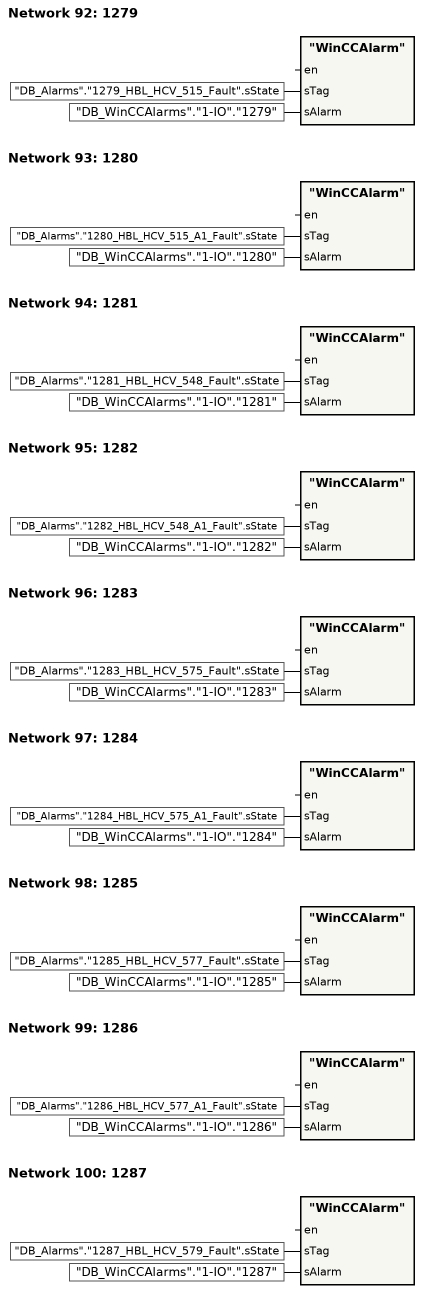
   "WinCCAlarm"(sTag := "DB_Alarms"."1279_HBL_HCV_515_Fault".sState, sAlarm := "DB_WinCCAlarms"."1-IO"."1279");
END_REGION

REGION Network 93: 1280
   "WinCCAlarm"(sTag := "DB_Alarms"."1280_HBL_HCV_515_A1_Fault".sState,
                sAlarm := "DB_WinCCAlarms"."1-IO"."1280");
END_REGION

REGION Network 94: 1281
   "WinCCAlarm"(sTag := "DB_Alarms"."1281_HBL_HCV_548_Fault".sState, sAlarm := "DB_WinCCAlarms"."1-IO"."1281");
END_REGION

REGION Network 95: 1282
   "WinCCAlarm"(sTag := "DB_Alarms"."1282_HBL_HCV_548_A1_Fault".sState,
                sAlarm := "DB_WinCCAlarms"."1-IO"."1282");
END_REGION

REGION Network 96: 1283
   "WinCCAlarm"(sTag := "DB_Alarms"."1283_HBL_HCV_575_Fault".sState, sAlarm := "DB_WinCCAlarms"."1-IO"."1283");
END_REGION

REGION Network 97: 1284
   "WinCCAlarm"(sTag := "DB_Alarms"."1284_HBL_HCV_575_A1_Fault".sState,
                sAlarm := "DB_WinCCAlarms"."1-IO"."1284");
END_REGION

REGION Network 98: 1285
   "WinCCAlarm"(sTag := "DB_Alarms"."1285_HBL_HCV_577_Fault".sState, sAlarm := "DB_WinCCAlarms"."1-IO"."1285");
END_REGION

REGION Network 99: 1286
   "WinCCAlarm"(sTag := "DB_Alarms"."1286_HBL_HCV_577_A1_Fault".sState,
                sAlarm := "DB_WinCCAlarms"."1-IO"."1286");
END_REGION

REGION Network 100: 1287
   "WinCCAlarm"(sTag := "DB_Alarms"."1287_HBL_HCV_579_Fault".sState, sAlarm := "DB_WinCCAlarms"."1-IO"."1287");
END_REGION

REGION Network 101: 1288
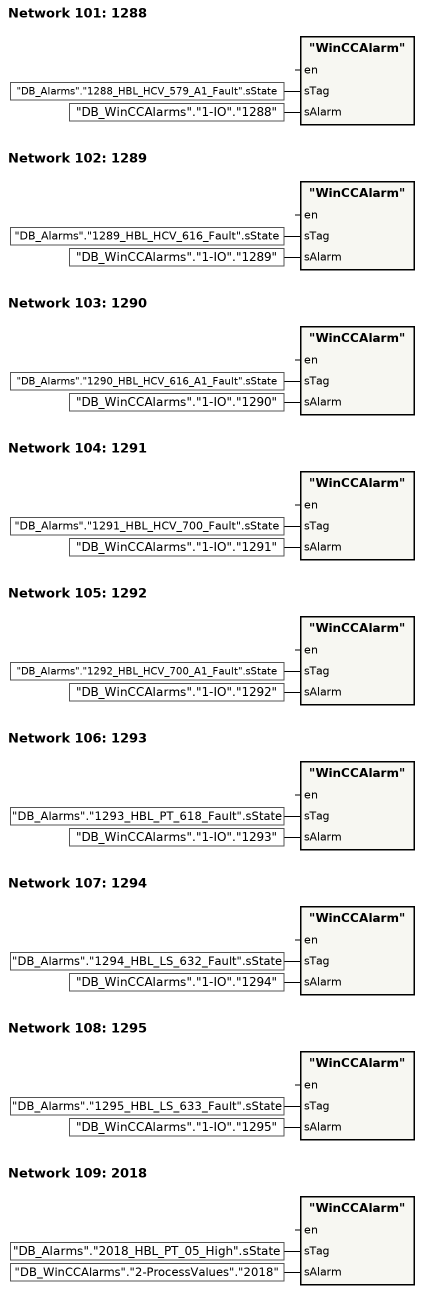
   "WinCCAlarm"(sTag := "DB_Alarms"."1288_HBL_HCV_579_A1_Fault".sState,
                sAlarm := "DB_WinCCAlarms"."1-IO"."1288");
END_REGION

REGION Network 102: 1289
   "WinCCAlarm"(sTag := "DB_Alarms"."1289_HBL_HCV_616_Fault".sState, sAlarm := "DB_WinCCAlarms"."1-IO"."1289");
END_REGION

REGION Network 103: 1290
   "WinCCAlarm"(sTag := "DB_Alarms"."1290_HBL_HCV_616_A1_Fault".sState,
                sAlarm := "DB_WinCCAlarms"."1-IO"."1290");
END_REGION

REGION Network 104: 1291
   "WinCCAlarm"(sTag := "DB_Alarms"."1291_HBL_HCV_700_Fault".sState, sAlarm := "DB_WinCCAlarms"."1-IO"."1291");
END_REGION

REGION Network 105: 1292
   "WinCCAlarm"(sTag := "DB_Alarms"."1292_HBL_HCV_700_A1_Fault".sState,
                sAlarm := "DB_WinCCAlarms"."1-IO"."1292");
END_REGION

REGION Network 106: 1293
   "WinCCAlarm"(sTag := "DB_Alarms"."1293_HBL_PT_618_Fault".sState, sAlarm := "DB_WinCCAlarms"."1-IO"."1293");
END_REGION

REGION Network 107: 1294
   "WinCCAlarm"(sTag := "DB_Alarms"."1294_HBL_LS_632_Fault".sState, sAlarm := "DB_WinCCAlarms"."1-IO"."1294");
END_REGION

REGION Network 108: 1295
   "WinCCAlarm"(sTag := "DB_Alarms"."1295_HBL_LS_633_Fault".sState, sAlarm := "DB_WinCCAlarms"."1-IO"."1295");
END_REGION

REGION Network 109: 2018
   "WinCCAlarm"(sTag := "DB_Alarms"."2018_HBL_PT_05_High".sState,
                sAlarm := "DB_WinCCAlarms"."2-ProcessValues"."2018");
END_REGION

REGION Network 110: 2028
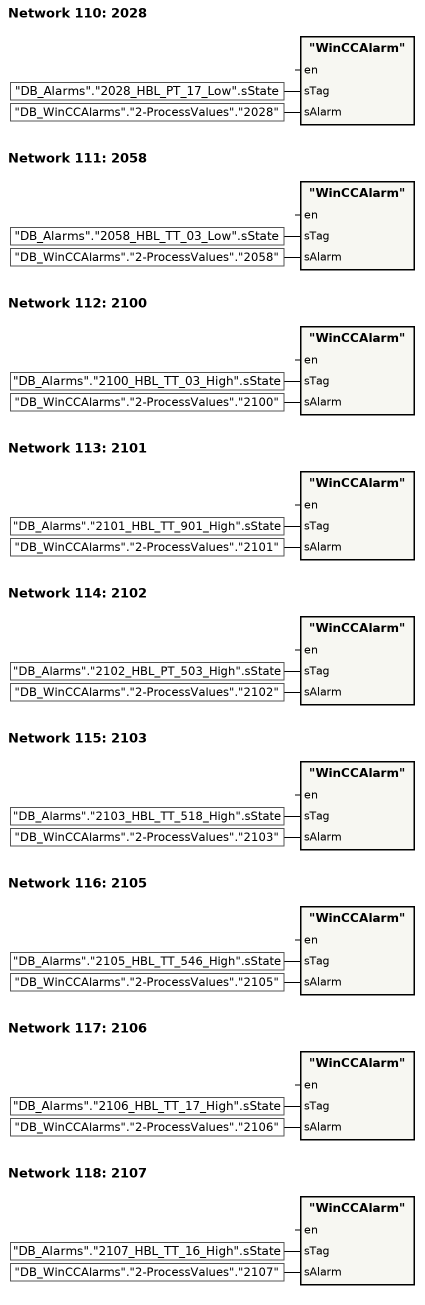
   "WinCCAlarm"(sTag := "DB_Alarms"."2028_HBL_PT_17_Low".sState,
                sAlarm := "DB_WinCCAlarms"."2-ProcessValues"."2028");
END_REGION

REGION Network 111: 2058
   "WinCCAlarm"(sTag := "DB_Alarms"."2058_HBL_TT_03_Low".sState,
                sAlarm := "DB_WinCCAlarms"."2-ProcessValues"."2058");
END_REGION

REGION Network 112: 2100
   "WinCCAlarm"(sTag := "DB_Alarms"."2100_HBL_TT_03_High".sState,
                sAlarm := "DB_WinCCAlarms"."2-ProcessValues"."2100");
END_REGION

REGION Network 113: 2101
   "WinCCAlarm"(sTag := "DB_Alarms"."2101_HBL_TT_901_High".sState,
                sAlarm := "DB_WinCCAlarms"."2-ProcessValues"."2101");
END_REGION

REGION Network 114: 2102
   "WinCCAlarm"(sTag := "DB_Alarms"."2102_HBL_PT_503_High".sState,
                sAlarm := "DB_WinCCAlarms"."2-ProcessValues"."2102");
END_REGION

REGION Network 115: 2103
   "WinCCAlarm"(sTag := "DB_Alarms"."2103_HBL_TT_518_High".sState,
                sAlarm := "DB_WinCCAlarms"."2-ProcessValues"."2103");
END_REGION

REGION Network 116: 2105
   "WinCCAlarm"(sTag := "DB_Alarms"."2105_HBL_TT_546_High".sState,
                sAlarm := "DB_WinCCAlarms"."2-ProcessValues"."2105");
END_REGION

REGION Network 117: 2106
   "WinCCAlarm"(sTag := "DB_Alarms"."2106_HBL_TT_17_High".sState,
                sAlarm := "DB_WinCCAlarms"."2-ProcessValues"."2106");
END_REGION

REGION Network 118: 2107
   "WinCCAlarm"(sTag := "DB_Alarms"."2107_HBL_TT_16_High".sState,
                sAlarm := "DB_WinCCAlarms"."2-ProcessValues"."2107");
END_REGION

REGION Network 119: 2108
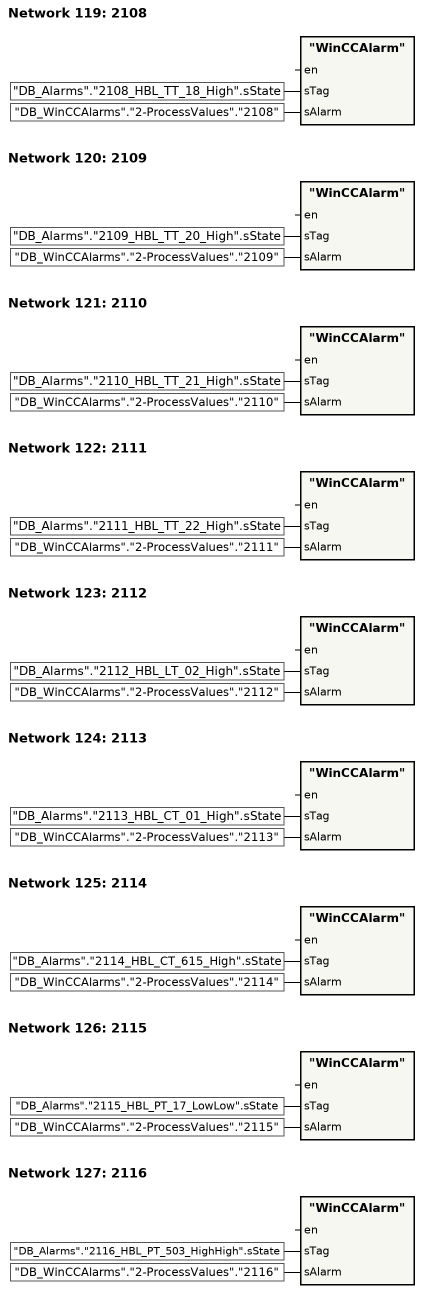
   "WinCCAlarm"(sTag := "DB_Alarms"."2108_HBL_TT_18_High".sState,
                sAlarm := "DB_WinCCAlarms"."2-ProcessValues"."2108");
END_REGION

REGION Network 120: 2109
   "WinCCAlarm"(sTag := "DB_Alarms"."2109_HBL_TT_20_High".sState,
                sAlarm := "DB_WinCCAlarms"."2-ProcessValues"."2109");
END_REGION

REGION Network 121: 2110
   "WinCCAlarm"(sTag := "DB_Alarms"."2110_HBL_TT_21_High".sState,
                sAlarm := "DB_WinCCAlarms"."2-ProcessValues"."2110");
END_REGION

REGION Network 122: 2111
   "WinCCAlarm"(sTag := "DB_Alarms"."2111_HBL_TT_22_High".sState,
                sAlarm := "DB_WinCCAlarms"."2-ProcessValues"."2111");
END_REGION

REGION Network 123: 2112
   "WinCCAlarm"(sTag := "DB_Alarms"."2112_HBL_LT_02_High".sState,
                sAlarm := "DB_WinCCAlarms"."2-ProcessValues"."2112");
END_REGION

REGION Network 124: 2113
   "WinCCAlarm"(sTag := "DB_Alarms"."2113_HBL_CT_01_High".sState,
                sAlarm := "DB_WinCCAlarms"."2-ProcessValues"."2113");
END_REGION

REGION Network 125: 2114
   "WinCCAlarm"(sTag := "DB_Alarms"."2114_HBL_CT_615_High".sState,
                sAlarm := "DB_WinCCAlarms"."2-ProcessValues"."2114");
END_REGION

REGION Network 126: 2115
   "WinCCAlarm"(sTag := "DB_Alarms"."2115_HBL_PT_17_LowLow".sState,
                sAlarm := "DB_WinCCAlarms"."2-ProcessValues"."2115");
END_REGION

REGION Network 127: 2116
   "WinCCAlarm"(sTag := "DB_Alarms"."2116_HBL_PT_503_HighHigh".sState,
                sAlarm := "DB_WinCCAlarms"."2-ProcessValues"."2116");
END_REGION

REGION Network 128: 2117
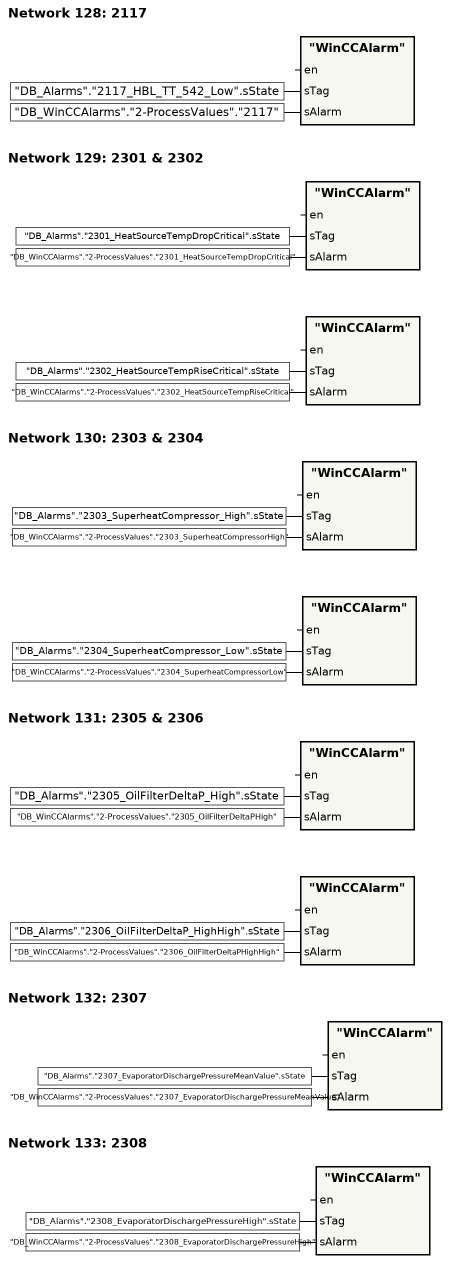
   "WinCCAlarm"(sTag := "DB_Alarms"."2117_HBL_TT_542_Low".sState,
                sAlarm := "DB_WinCCAlarms"."2-ProcessValues"."2117");
END_REGION

REGION Network 129: 2301 & 2302
   "WinCCAlarm"(sTag := "DB_Alarms"."2301_HeatSourceTempDropCritical".sState,
                sAlarm := "DB_WinCCAlarms"."2-ProcessValues"."2301_HeatSourceTempDropCritical");
   "WinCCAlarm"(sTag := "DB_Alarms"."2302_HeatSourceTempRiseCritical".sState,
                sAlarm := "DB_WinCCAlarms"."2-ProcessValues"."2302_HeatSourceTempRiseCritical");
END_REGION

REGION Network 130: 2303 & 2304
   "WinCCAlarm"(sTag := "DB_Alarms"."2303_SuperheatCompressor_High".sState,
                sAlarm := "DB_WinCCAlarms"."2-ProcessValues"."2303_SuperheatCompressorHigh");
   "WinCCAlarm"(sTag := "DB_Alarms"."2304_SuperheatCompressor_Low".sState,
                sAlarm := "DB_WinCCAlarms"."2-ProcessValues"."2304_SuperheatCompressorLow");
END_REGION

REGION Network 131: 2305 & 2306
   "WinCCAlarm"(sTag := "DB_Alarms"."2305_OilFilterDeltaP_High".sState,
                sAlarm := "DB_WinCCAlarms"."2-ProcessValues"."2305_OilFilterDeltaPHigh");
   "WinCCAlarm"(sTag := "DB_Alarms"."2306_OilFilterDeltaP_HighHigh".sState,
                sAlarm := "DB_WinCCAlarms"."2-ProcessValues"."2306_OilFilterDeltaPHighHigh");
END_REGION

REGION Network 132: 2307
   "WinCCAlarm"(sTag := "DB_Alarms"."2307_EvaporatorDischargePressureMeanValue".sState,
                sAlarm := "DB_WinCCAlarms"."2-ProcessValues"."2307_EvaporatorDischargePressureMeanValue");
END_REGION

REGION Network 133: 2308
   "WinCCAlarm"(sTag := "DB_Alarms"."2308_EvaporatorDischargePressureHigh".sState,
                sAlarm := "DB_WinCCAlarms"."2-ProcessValues"."2308_EvaporatorDischargePressureHigh");
END_REGION

REGION Network 134: 2309
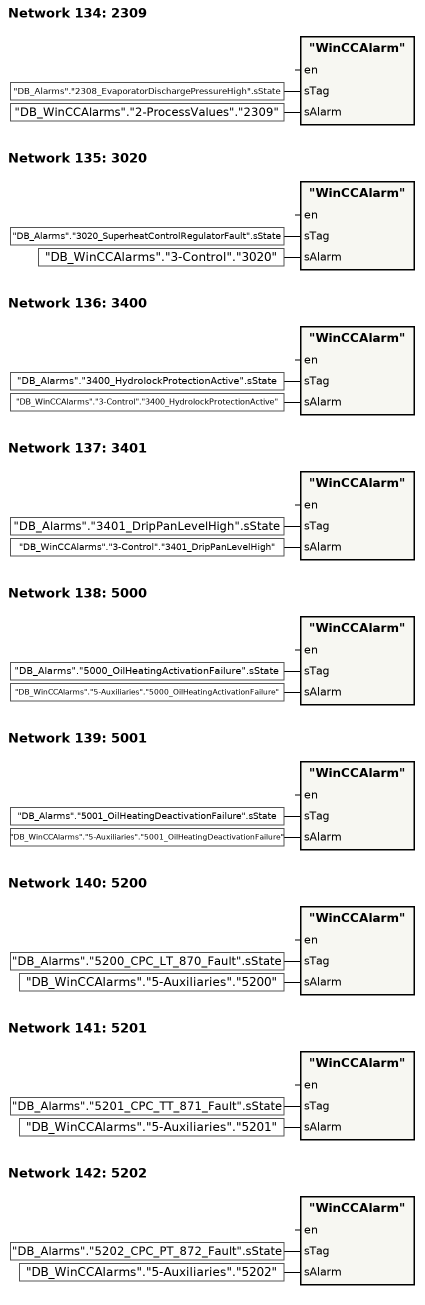
   "WinCCAlarm"(sTag := "DB_Alarms"."2308_EvaporatorDischargePressureHigh".sState,
                sAlarm := "DB_WinCCAlarms"."2-ProcessValues"."2309");
END_REGION

REGION Network 135: 3020
   "WinCCAlarm"(sTag := "DB_Alarms"."3020_SuperheatControlRegulatorFault".sState,
                sAlarm := "DB_WinCCAlarms"."3-Control"."3020");
END_REGION

REGION Network 136: 3400
   "WinCCAlarm"(sTag := "DB_Alarms"."3400_HydrolockProtectionActive".sState,
                sAlarm := "DB_WinCCAlarms"."3-Control"."3400_HydrolockProtectionActive");
END_REGION

REGION Network 137: 3401
   "WinCCAlarm"(sTag := "DB_Alarms"."3401_DripPanLevelHigh".sState,
                sAlarm := "DB_WinCCAlarms"."3-Control"."3401_DripPanLevelHigh");
END_REGION

REGION Network 138: 5000
   "WinCCAlarm"(sTag := "DB_Alarms"."5000_OilHeatingActivationFailure".sState,
                sAlarm := "DB_WinCCAlarms"."5-Auxiliaries"."5000_OilHeatingActivationFailure");
END_REGION

REGION Network 139: 5001
   "WinCCAlarm"(sTag := "DB_Alarms"."5001_OilHeatingDeactivationFailure".sState,
                sAlarm := "DB_WinCCAlarms"."5-Auxiliaries"."5001_OilHeatingDeactivationFailure");
END_REGION

REGION Network 140: 5200
   "WinCCAlarm"(sTag := "DB_Alarms"."5200_CPC_LT_870_Fault".sState,
                sAlarm := "DB_WinCCAlarms"."5-Auxiliaries"."5200");
END_REGION

REGION Network 141: 5201
   "WinCCAlarm"(sTag := "DB_Alarms"."5201_CPC_TT_871_Fault".sState,
                sAlarm := "DB_WinCCAlarms"."5-Auxiliaries"."5201");
END_REGION

REGION Network 142: 5202
   "WinCCAlarm"(sTag := "DB_Alarms"."5202_CPC_PT_872_Fault".sState,
                sAlarm := "DB_WinCCAlarms"."5-Auxiliaries"."5202");
END_REGION

REGION Network 143: 5203
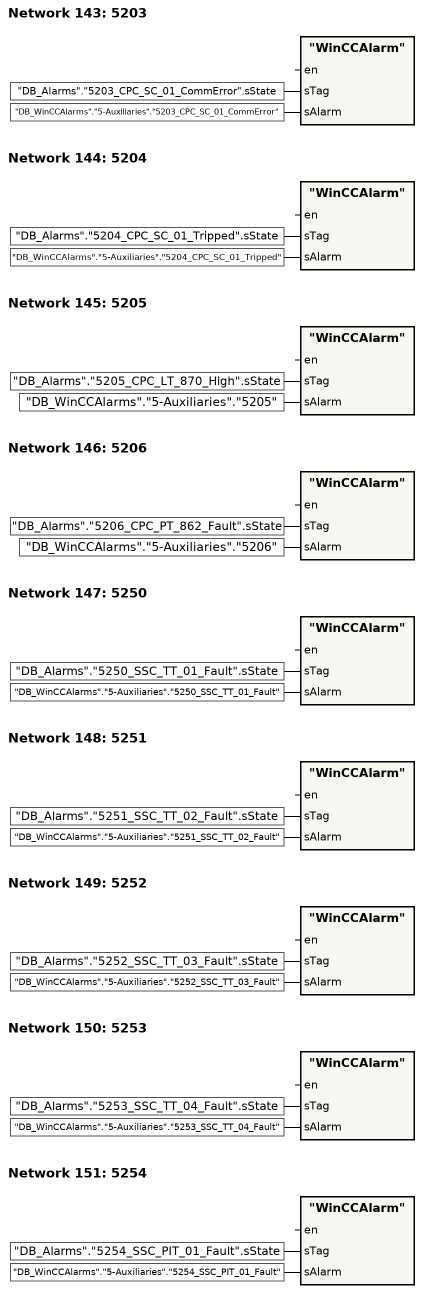
   "WinCCAlarm"(sTag := "DB_Alarms"."5203_CPC_SC_01_CommError".sState,
                sAlarm := "DB_WinCCAlarms"."5-Auxiliaries"."5203_CPC_SC_01_CommError");
END_REGION

REGION Network 144: 5204
   "WinCCAlarm"(sTag := "DB_Alarms"."5204_CPC_SC_01_Tripped".sState,
                sAlarm := "DB_WinCCAlarms"."5-Auxiliaries"."5204_CPC_SC_01_Tripped");
END_REGION

REGION Network 145: 5205
   "WinCCAlarm"(sTag := "DB_Alarms"."5205_CPC_LT_870_High".sState,
                sAlarm := "DB_WinCCAlarms"."5-Auxiliaries"."5205");
END_REGION

REGION Network 146: 5206
   "WinCCAlarm"(sTag := "DB_Alarms"."5206_CPC_PT_862_Fault".sState,
                sAlarm := "DB_WinCCAlarms"."5-Auxiliaries"."5206");
END_REGION

REGION Network 147: 5250
   "WinCCAlarm"(sTag := "DB_Alarms"."5250_SSC_TT_01_Fault".sState,
                sAlarm := "DB_WinCCAlarms"."5-Auxiliaries"."5250_SSC_TT_01_Fault");
END_REGION

REGION Network 148: 5251
   "WinCCAlarm"(sTag := "DB_Alarms"."5251_SSC_TT_02_Fault".sState,
                sAlarm := "DB_WinCCAlarms"."5-Auxiliaries"."5251_SSC_TT_02_Fault");
END_REGION

REGION Network 149: 5252
   "WinCCAlarm"(sTag := "DB_Alarms"."5252_SSC_TT_03_Fault".sState,
                sAlarm := "DB_WinCCAlarms"."5-Auxiliaries"."5252_SSC_TT_03_Fault");
END_REGION

REGION Network 150: 5253
   "WinCCAlarm"(sTag := "DB_Alarms"."5253_SSC_TT_04_Fault".sState,
                sAlarm := "DB_WinCCAlarms"."5-Auxiliaries"."5253_SSC_TT_04_Fault");
END_REGION

REGION Network 151: 5254
   "WinCCAlarm"(sTag := "DB_Alarms"."5254_SSC_PIT_01_Fault".sState,
                sAlarm := "DB_WinCCAlarms"."5-Auxiliaries"."5254_SSC_PIT_01_Fault");
END_REGION

REGION Network 152: 5255
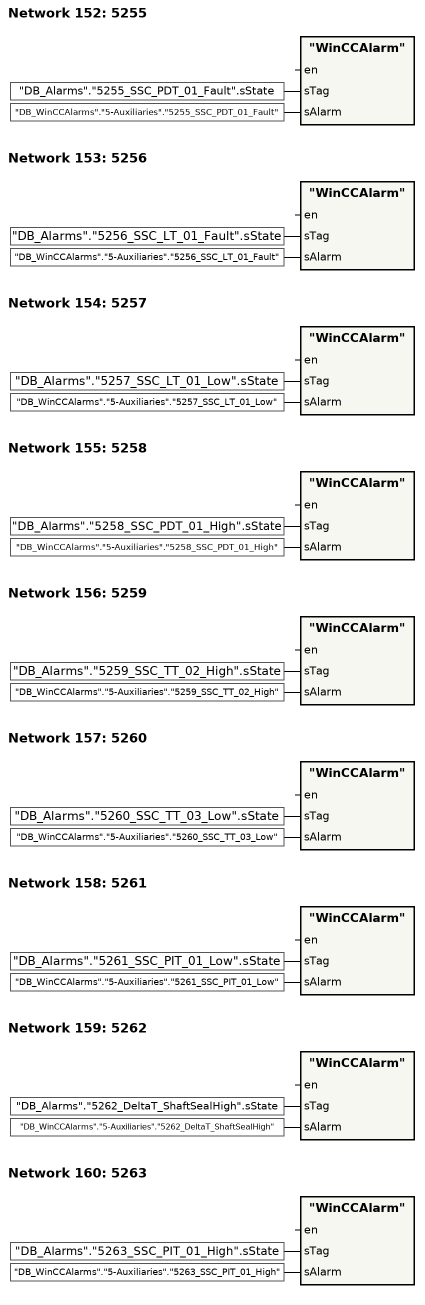
   "WinCCAlarm"(sTag := "DB_Alarms"."5255_SSC_PDT_01_Fault".sState,
                sAlarm := "DB_WinCCAlarms"."5-Auxiliaries"."5255_SSC_PDT_01_Fault");
END_REGION

REGION Network 153: 5256
   "WinCCAlarm"(sTag := "DB_Alarms"."5256_SSC_LT_01_Fault".sState,
                sAlarm := "DB_WinCCAlarms"."5-Auxiliaries"."5256_SSC_LT_01_Fault");
END_REGION

REGION Network 154: 5257
   "WinCCAlarm"(sTag := "DB_Alarms"."5257_SSC_LT_01_Low".sState,
                sAlarm := "DB_WinCCAlarms"."5-Auxiliaries"."5257_SSC_LT_01_Low");
END_REGION

REGION Network 155: 5258
   "WinCCAlarm"(sTag := "DB_Alarms"."5258_SSC_PDT_01_High".sState,
                sAlarm := "DB_WinCCAlarms"."5-Auxiliaries"."5258_SSC_PDT_01_High");
END_REGION

REGION Network 156: 5259
   "WinCCAlarm"(sTag := "DB_Alarms"."5259_SSC_TT_02_High".sState,
                sAlarm := "DB_WinCCAlarms"."5-Auxiliaries"."5259_SSC_TT_02_High");
END_REGION

REGION Network 157: 5260
   "WinCCAlarm"(sTag := "DB_Alarms"."5260_SSC_TT_03_Low".sState,
                sAlarm := "DB_WinCCAlarms"."5-Auxiliaries"."5260_SSC_TT_03_Low");
END_REGION

REGION Network 158: 5261
   "WinCCAlarm"(sTag := "DB_Alarms"."5261_SSC_PIT_01_Low".sState,
                sAlarm := "DB_WinCCAlarms"."5-Auxiliaries"."5261_SSC_PIT_01_Low");
END_REGION

REGION Network 159: 5262
   "WinCCAlarm"(sTag := "DB_Alarms"."5262_DeltaT_ShaftSealHigh".sState,
                sAlarm := "DB_WinCCAlarms"."5-Auxiliaries"."5262_DeltaT_ShaftSealHigh");
END_REGION

REGION Network 160: 5263
   "WinCCAlarm"(sTag := "DB_Alarms"."5263_SSC_PIT_01_High".sState,
                sAlarm := "DB_WinCCAlarms"."5-Auxiliaries"."5263_SSC_PIT_01_High");
END_REGION

REGION Network 161: 5268
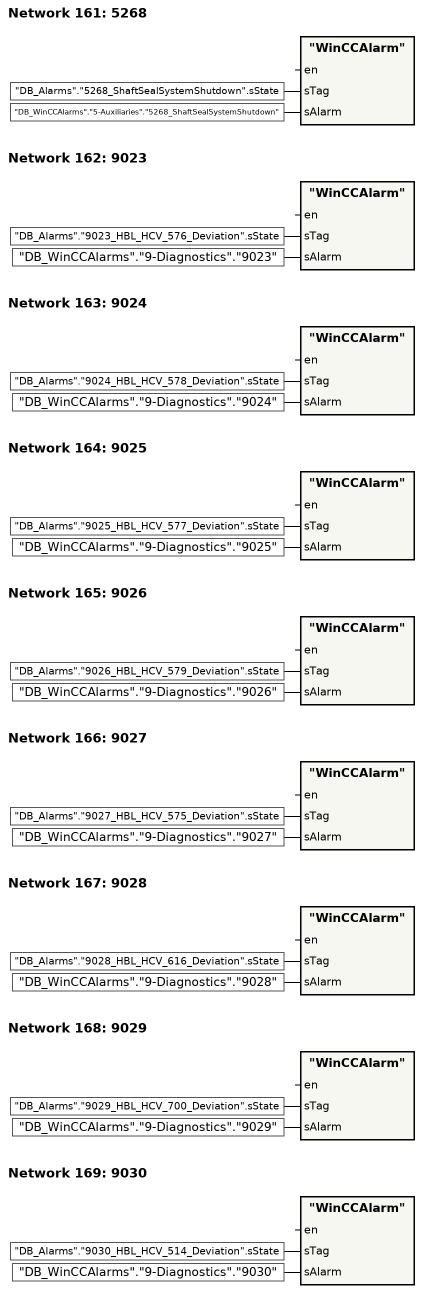
   "WinCCAlarm"(sTag := "DB_Alarms"."5268_ShaftSealSystemShutdown".sState,
                sAlarm := "DB_WinCCAlarms"."5-Auxiliaries"."5268_ShaftSealSystemShutdown");
END_REGION

REGION Network 162: 9023
   "WinCCAlarm"(sTag := "DB_Alarms"."9023_HBL_HCV_576_Deviation".sState,
                sAlarm := "DB_WinCCAlarms"."9-Diagnostics"."9023");
END_REGION

REGION Network 163: 9024
   "WinCCAlarm"(sTag := "DB_Alarms"."9024_HBL_HCV_578_Deviation".sState,
                sAlarm := "DB_WinCCAlarms"."9-Diagnostics"."9024");
END_REGION

REGION Network 164: 9025
   "WinCCAlarm"(sTag := "DB_Alarms"."9025_HBL_HCV_577_Deviation".sState,
                sAlarm := "DB_WinCCAlarms"."9-Diagnostics"."9025");
END_REGION

REGION Network 165: 9026
   "WinCCAlarm"(sTag := "DB_Alarms"."9026_HBL_HCV_579_Deviation".sState,
                sAlarm := "DB_WinCCAlarms"."9-Diagnostics"."9026");
END_REGION

REGION Network 166: 9027
   "WinCCAlarm"(sTag := "DB_Alarms"."9027_HBL_HCV_575_Deviation".sState,
                sAlarm := "DB_WinCCAlarms"."9-Diagnostics"."9027");
END_REGION

REGION Network 167: 9028
   "WinCCAlarm"(sTag := "DB_Alarms"."9028_HBL_HCV_616_Deviation".sState,
                sAlarm := "DB_WinCCAlarms"."9-Diagnostics"."9028");
END_REGION

REGION Network 168: 9029
   "WinCCAlarm"(sTag := "DB_Alarms"."9029_HBL_HCV_700_Deviation".sState,
                sAlarm := "DB_WinCCAlarms"."9-Diagnostics"."9029");
END_REGION

REGION Network 169: 9030
   "WinCCAlarm"(sTag := "DB_Alarms"."9030_HBL_HCV_514_Deviation".sState,
                sAlarm := "DB_WinCCAlarms"."9-Diagnostics"."9030");
END_REGION

REGION Network 170: 9031
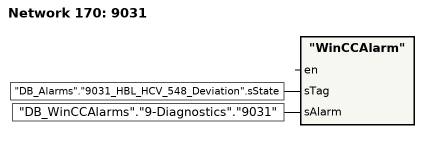
   "WinCCAlarm"(sTag := "DB_Alarms"."9031_HBL_HCV_548_Deviation".sState,
                sAlarm := "DB_WinCCAlarms"."9-Diagnostics"."9031");
END_REGION
END_FUNCTION

FUNCTION "WinCCAlarm" : Void   // FC13, FBD
{ S7_Optimized_Access := 'TRUE' }
VERSION : 0.1
// stored: AutoNumber true, IsIECCheckEnabled false, SetENOAutomatically false, UDAEnableTagReadback false
   VAR_IN_OUT
      sTag : "stAlarmState";   // OPC alarm object
      sAlarm : "stWinCCAlarm";   // WinCC alarm object
   END_VAR
BEGIN

REGION Network 1 (SCL): WinCC alarm object
   // Possible alarm states:
   // bActive | bActiveUnack | State                                        | Show in Wincc alarm list? | Behaviour
   //-----------------------------------------------------------------------------------------------------------------------------------
   //    0    |      0       | No alarm                                     | No alarm                  | Nothing
   //    1    |      1       | Unacknowledged and active alarm condition    | Alarm                     | Stays on screen when acknowledged
   //    1    |      0       | Acknowledged and active alarm condition      | Alarm                     | Disappears when condition goes away
   //    0    1      1       | Unacknowledged and alarm condition is gone   | Alarm                     | Stays on screen until acknowledged

   #sAlarm.Memory.%X0 := #sTag.bActive OR #sTag.bActiveUnack;
END_REGION
END_FUNCTION

FUNCTION_BLOCK "ApplicationCommunication"   // FB6, LAD
{ S7_Optimized_Access := 'TRUE' }
VERSION : 0.1
// Note some networks are in Ladder because the FBD equivalents are too bulky and the SCL equivalents are too easy to screw up accidentally.
// stored: AutoNumber true, IsIECCheckEnabled false, IsRetainMemResEnabled false, MemoryReserve 0, SetENOAutomatically false, UDAEnableTagReadback false
   VAR
      ExpansionRegulatorManualOn { ExternalAccessible := 'False'; ExternalVisible := 'False'; ExternalWritable := 'False'} : Bool;
      ExpansionRegulatorManualOff { ExternalAccessible := 'False'; ExternalVisible := 'False'; ExternalWritable := 'False'; S7_SetPoint := 'True'} : Bool;
      HeatSinkOutManualOn { ExternalAccessible := 'False'; ExternalVisible := 'False'; ExternalWritable := 'False'} : Bool;
      HeatSinkOutManualOff { ExternalAccessible := 'False'; ExternalVisible := 'False'; ExternalWritable := 'False'} : Bool;
      PerformanceManualModeOn { ExternalAccessible := 'False'; ExternalVisible := 'False'; ExternalWritable := 'False'} : Bool;
      PerformanceManualModeOff { ExternalAccessible := 'False'; ExternalVisible := 'False'; ExternalWritable := 'False'} : Bool;
      OilHeatingManualOn { ExternalAccessible := 'False'; ExternalVisible := 'False'; ExternalWritable := 'False'} : Bool;
      OilHeatingManualOff { ExternalAccessible := 'False'; ExternalVisible := 'False'; ExternalWritable := 'False'} : Bool;
      PinchManualModeOn { ExternalAccessible := 'False'; ExternalVisible := 'False'; ExternalWritable := 'False'} : Bool;
      PinchManualModeOff { ExternalAccessible := 'False'; ExternalVisible := 'False'; ExternalWritable := 'False'} : Bool;
      SuperheatManualOn { ExternalAccessible := 'False'; ExternalVisible := 'False'; ExternalWritable := 'False'} : Bool;
      SuperheatManualOff { ExternalAccessible := 'False'; ExternalVisible := 'False'; ExternalWritable := 'False'} : Bool;
      AlarmAckOn { ExternalAccessible := 'False'; ExternalVisible := 'False'; ExternalWritable := 'False'} : Bool;
      AlarmAckOff { ExternalAccessible := 'False'; ExternalVisible := 'False'; ExternalWritable := 'False'} : Bool;
      ResetEstopOn { ExternalAccessible := 'False'; ExternalVisible := 'False'; ExternalWritable := 'False'} : Bool;
      ResetEstopOff { ExternalAccessible := 'False'; ExternalVisible := 'False'; ExternalWritable := 'False'} : Bool;
      FastStopOn { ExternalAccessible := 'False'; ExternalVisible := 'False'; ExternalWritable := 'False'} : Bool;
      ExpansionManualPrev { ExternalAccessible := 'False'; ExternalVisible := 'False'; ExternalWritable := 'False'} : Real;
      HeatSinkManualPrev { ExternalAccessible := 'False'; ExternalVisible := 'False'; ExternalWritable := 'False'} : Real;
      PerformanceManualPrev { ExternalAccessible := 'False'; ExternalVisible := 'False'; ExternalWritable := 'False'} : Real;
      OilHeatingManualPrev { ExternalAccessible := 'False'; ExternalVisible := 'False'; ExternalWritable := 'False'} : Real;
      PinchManualPrev { ExternalAccessible := 'False'; ExternalVisible := 'False'; ExternalWritable := 'False'} : Real;
      SuperheatManualPrev { ExternalAccessible := 'False'; ExternalVisible := 'False'; ExternalWritable := 'False'} : Real;
      HeatboosterSetpointPrev { ExternalAccessible := 'False'; ExternalVisible := 'False'; ExternalWritable := 'False'} : Real;
      RegulationTargetPrev { ExternalAccessible := 'False'; ExternalVisible := 'False'; ExternalWritable := 'False'} : Int;
      S7Watchdog : "fbHeartbeatCount2";
   END_VAR
   VAR_TEMP
      bDummy : Bool;
      fDummy : Real;
   END_VAR
   VAR_TEMP   // added for the SCL form of the ladder/FBD networks
      _w1 : Bool;
      _w2 : Bool;
      _w3 : Bool;
      _w4 : Bool;
      _w5 : Bool;
      _w6 : Bool;
      _w7 : Bool;
      _w8 : Bool;
      _w9 : Bool;
      _w10 : Bool;
   END_VAR
BEGIN

REGION Network 1 (SCL): Status
   // Applications PLC GETs these.
   "DB_Application".FromHB.EmergencyStop       := "DB_System".bEmergencyStop;
   "DB_Application".FromHB.OilHeatersGroup1    := "DB_DO".HBL_EC_01;
   "DB_Application".FromHB.OilHeatersGroup2    := "DB_DO".HBL_EC_02;
   "DB_Application".FromHB.HBL_SC_10_Ready     := "DB_InverterDrives".HBL_SC_10.Stat.bReady;
   "DB_Application".FromHB.HBL_SC_10_Run       := "DB_InverterDrives".HBL_SC_10.Stat.bRun;
   "DB_Application".FromHB.HBL_HV_630           := "DB_DO".HBL_HV_630;
   "DB_Application".FromHB.CPC_P_01            := "DB_DO".CPC_P_01;
   "DB_Application".FromHB.SSC_P_01            := "DB_DO".SSC_P_01;
   "DB_Application".FromHB.HBL_SC_10_Tripped   := "DB_InverterDrives".HBL_SC_10.Stat.bTrip;
   "DB_Application".FromHB.HBL_SC_02_Ready     := "DB_InverterDrives".HBL_SC_02.Stat.bReady;
   "DB_Application".FromHB.HBL_SC_02_Run       := "DB_InverterDrives".HBL_SC_02.Stat.bRun;
   "DB_Application".FromHB.HBL_SC_02_Tripped   := "DB_InverterDrives".HBL_SC_02.Stat.bTrip;
   "DB_Application".FromHB.SSC_F_01            := "DB_DO".SSC_F_01;
   "DB_Application".FromHB.SSC_P_02            := "DB_DO".SSC_P_02;
   "DB_Application".FromHB.HBL_LS_01           := "DB_DI".HBL_LS_01.bValue;
   "DB_Application".FromHB.HBL_LS_02           := "DB_DI".HBL_LS_02.bValue;
   "DB_Application".FromHB.MachineState        := "DB_State".State.State_Number;
   "DB_Application".FromHB.CompressorType      := "DB_CurrentSetting".Compressor.CompressorTypeNumber;
   "DB_Application".FromHB.SystemType          := "DB_CurrentSetting".System.SystemTypeNumber;
   "DB_Application".FromHB.RefrigerantType     := "DB_CurrentSetting".Fluid.FluidTypeNumber;
   "DB_Application".FromHB.UptimeHours         := UDINT_TO_INT("DB_System".SystemUptime.nHours);
   "DB_Application".FromHB.UptimeMinutes       := "DB_System".SystemUptime.nMinutes;
   "DB_Application".FromHB.UptimeSeconds       := "DB_System".SystemUptime.nSeconds;
   "DB_Application".FromHB.ActiveTimeHours     := UDINT_TO_INT("DB_System".SystemActiveTime.nHours);
   "DB_Application".FromHB.ActiveTimeMinutes   := "DB_System".SystemActiveTime.nMinutes;
   "DB_Application".FromHB.ActiveTimeSeconds   := "DB_System".SystemActiveTime.nSeconds;
   "DB_Application".FromHB.RunningTimeHours    := UDINT_TO_INT("DB_System".RunningTime.nHours);
   "DB_Application".FromHB.RunningTimeMinutes  := "DB_System".RunningTime.nMinutes;
   "DB_Application".FromHB.RunningTimeSeconds  := "DB_System".RunningTime.nSeconds;
   "DB_Application".FromHB.HeatboosterSetpoint := "DB_Regulators".HeatboosterSetpoint;
   "DB_Application".FromHB.RegulationTarget    := "DB_Regulators".RegulationTarget;
   "DB_Application".FromHB.HBL_HCV_514_Force   := FALSE; // ###FIX
   "DB_Application".FromHB.HBL_HCV_514         := 5.14; //##FIX
   "DB_Application".FromHB.HBL_HCV_548_Force   := FALSE; // ##FIX
   "DB_Application".FromHB.HBL_HCV_548         := 5.48; //##FIX
END_REGION

REGION Network 2 (SCL): DB_AI
   // Copy only .fValues for minimum bandwidth
   "DB_Application".FromHB.DB_AI.HBL_TT_502 := "DB_AI".HBL_TT_502.Eng.fValue;
   "DB_Application".FromHB.DB_AI.HBL_PT_503 := "DB_AI".HBL_PT_503.Eng.fValue;
   "DB_Application".FromHB.DB_AI.HBL_TT_504 := "DB_AI".HBL_TT_504.Eng.fValue;
   "DB_Application".FromHB.DB_AI.HBL_LT_510 := "DB_AI".HBL_LT_510.Eng.fValue;
   "DB_Application".FromHB.DB_AI.HBL_PT_511 := "DB_AI".HBL_PT_511.Eng.fValue;
   "DB_Application".FromHB.DB_AI.HBL_TT_512 := "DB_AI".HBL_TT_512.Eng.fValue;
   "DB_Application".FromHB.DB_AI.HBL_TT_516 := "DB_AI".HBL_TT_516.Eng.fValue;
   "DB_Application".FromHB.DB_AI.HBL_PT_517 := "DB_AI".HBL_PT_517.Eng.fValue;
   "DB_Application".FromHB.DB_AI.HBL_TT_518 := "DB_AI".HBL_TT_518.Eng.fValue;
   "DB_Application".FromHB.DB_AI.HBL_PT_519 := "DB_AI".HBL_PT_519.Eng.fValue;
   "DB_Application".FromHB.DB_AI.HBL_FT_520 := "DB_AI".HBL_FT_520.Eng.fValue;
   "DB_Application".FromHB.DB_AI.HBL_TT_530 := "DB_AI".HBL_TT_530.Eng.fValue;
   "DB_Application".FromHB.DB_AI.HBL_PT_531 := "DB_AI".HBL_PT_531.Eng.fValue;
   "DB_Application".FromHB.DB_AI.HBL_TT_532 := "DB_AI".HBL_TT_532.Eng.fValue;
   "DB_Application".FromHB.DB_AI.HBL_TT_533 := "DB_AI".HBL_TT_533.Eng.fValue;
   "DB_Application".FromHB.DB_AI.HBL_PT_534 := "DB_AI".HBL_PT_534.Eng.fValue;
   "DB_Application".FromHB.DB_AI.HBL_AT_535 := "DB_AI".HBL_AT_535.Eng.fValue;
   "DB_Application".FromHB.DB_AI.HBL_TT_540 := "DB_AI".HBL_TT_540.Eng.fValue;
   "DB_Application".FromHB.DB_AI.HBL_PT_541 := "DB_AI".HBL_PT_541.Eng.fValue;
   "DB_Application".FromHB.DB_AI.HBL_TT_542 := "DB_AI".HBL_TT_542.Eng.fValue;
   "DB_Application".FromHB.DB_AI.HBL_TT_543 := "DB_AI".HBL_TT_543.Eng.fValue;
   "DB_Application".FromHB.DB_AI.HBL_PT_544 := "DB_AI".HBL_PT_544.Eng.fValue;
   "DB_Application".FromHB.DB_AI.HBL_AT_545 := "DB_AI".HBL_AT_545.Eng.fValue;
   "DB_Application".FromHB.DB_AI.HBL_TT_546 := "DB_AI".HBL_TT_546.Eng.fValue;
   "DB_Application".FromHB.DB_AI.HBL_PT_547 := "DB_AI".HBL_PT_547.Eng.fValue;
   "DB_Application".FromHB.DB_AI.HBL_TT_571 := "DB_AI".HBL_TT_571.Eng.fValue;
   "DB_Application".FromHB.DB_AI.HBL_PT_572 := "DB_AI".HBL_PT_572.Eng.fValue;
   "DB_Application".FromHB.DB_AI.HBL_TT_573 := "DB_AI".HBL_TT_573.Eng.fValue;
   "DB_Application".FromHB.DB_AI.HBL_LT_610 := "DB_AI".HBL_LT_610.Eng.fValue;
   "DB_Application".FromHB.DB_AI.HBL_TT_611 := "DB_AI".HBL_TT_611.Eng.fValue;
   "DB_Application".FromHB.DB_AI.HBL_PT_612 := "DB_AI".HBL_PT_612.Eng.fValue;
   "DB_Application".FromHB.DB_AI.HBL_CT_615 := "DB_AI".HBL_CT_615.Eng.fValue;
   "DB_Application".FromHB.DB_AI.HBL_PT_618 := "DB_AI".HBL_PT_618.Eng.fValue;
   "DB_Application".FromHB.DB_AI.HBL_PT_635 := "DB_AI".HBL_PT_635.Eng.fValue;
   "DB_Application".FromHB.DB_AI.HBL_PT_636 := "DB_AI".HBL_PT_636.Eng.fValue;
   "DB_Application".FromHB.DB_AI.HBL_LT_650 := "DB_AI".HBL_LT_650.Eng.fValue;
   "DB_Application".FromHB.DB_AI.HBL_PT_651 := "DB_AI".HBL_PT_651.Eng.fValue;
   "DB_Application".FromHB.DB_AI.HBL_PT_701 := "DB_AI".HBL_PT_701.Eng.fValue;
   "DB_Application".FromHB.DB_AI.HBL_PT_702 := "DB_AI".HBL_PT_702.Eng.fValue;
   "DB_Application".FromHB.DB_AI.HBL_PT_703 := "DB_AI".HBL_PT_703.Eng.fValue;

   "DB_Application".FromHB.DB_AI.CPC_LT_870 := "DB_AI".CPC_LT_870.Eng.fValue;
   "DB_Application".FromHB.DB_AI.CPC_TT_871 := "DB_AI".CPC_TT_871.Eng.fValue;
   "DB_Application".FromHB.DB_AI.CPC_PT_872 := "DB_AI".CPC_PT_872.Eng.fValue;
   "DB_Application".FromHB.DB_AI.CPC_PT_862 := "DB_AI".CPC_PT_862.Eng.fValue;
   "DB_Application".FromHB.DB_AI.HBL_TT_901 := "DB_AI".HBL_TT_901.Eng.fValue;
   "DB_Application".FromHB.DB_AI.HBL_PT_902 := "DB_AI".HBL_PT_902.Eng.fValue;

   "DB_Application".FromHB.DB_AI.HBL_TT_03 := "DB_AI".HBL_TT_03.Eng.fValue;
   "DB_Application".FromHB.DB_AI.HBL_TT_16 := "DB_AI".HBL_TT_16.Eng.fValue;
   "DB_Application".FromHB.DB_AI.HBL_TT_17 := "DB_AI".HBL_TT_17.Eng.fValue;
   "DB_Application".FromHB.DB_AI.HBL_TT_18 := "DB_AI".HBL_TT_18.Eng.fValue;
   "DB_Application".FromHB.DB_AI.HBL_TT_20 := "DB_AI".HBL_TT_20.Eng.fValue;
   "DB_Application".FromHB.DB_AI.HBL_TT_21 := "DB_AI".HBL_TT_21.Eng.fValue;
   "DB_Application".FromHB.DB_AI.HBL_TT_22 := "DB_AI".HBL_TT_22.Eng.fValue;
   "DB_Application".FromHB.DB_AI.HBL_TT_23 := "DB_AI".HBL_TT_23.Eng.fValue;
   "DB_Application".FromHB.DB_AI.HBL_TT_24 := "DB_AI".HBL_TT_24.Eng.fValue;
   "DB_Application".FromHB.DB_AI.HBL_TT_25 := "DB_AI".HBL_TT_25.Eng.fValue;
   "DB_Application".FromHB.DB_AI.HBL_TT_26 := "DB_AI".HBL_TT_26.Eng.fValue;
   "DB_Application".FromHB.DB_AI.HBL_TT_27 := "DB_AI".HBL_TT_27.Eng.fValue;
   "DB_Application".FromHB.DB_AI.HBL_PT_05 := "DB_AI".HBL_PT_05.Eng.fValue;
   "DB_Application".FromHB.DB_AI.HBL_PT_06 := "DB_AI".HBL_PT_960.Eng.fValue;
   "DB_Application".FromHB.DB_AI.HBL_PT_17 := "DB_AI".HBL_PT_961.Eng.fValue;
   "DB_Application".FromHB.DB_AI.HBL_CT_01 := "DB_AI".HBL_CT_01.Eng.fValue;
   "DB_Application".FromHB.DB_AI.HBL_CT_03 := "DB_AI".HBL_CT_950.Eng.fValue;

   "DB_Application".FromHB.DB_AI.SSC_TT_01 := "DB_AI".SSC_TT_01.Eng.fValue;
   "DB_Application".FromHB.DB_AI.SSC_TT_02 := "DB_AI".SSC_TT_02.Eng.fValue;
   "DB_Application".FromHB.DB_AI.SSC_TT_03 := "DB_AI".SSC_TT_03.Eng.fValue;
   "DB_Application".FromHB.DB_AI.SSC_TT_04 := "DB_AI".SSC_TT_04.Eng.fValue;
   "DB_Application".FromHB.DB_AI.SSC_PIT_01 := "DB_AI".SSC_PIT_01.Eng.fValue;
   "DB_Application".FromHB.DB_AI.SSC_PDT_01 := "DB_AI".SSC_PDT_01.Eng.fValue;
   "DB_Application".FromHB.DB_AI.SSC_LT_01 := "DB_AI".SSC_LT_01.Eng.fValue;
END_REGION

REGION Network 3 (SCL): DB_Calc
   // Done this way for minimum bandwidth
   "DB_Application".FromHB.DB_Calc.Compressor_CrankcaseSaturationTemperature   := "DB_Calc".Compressor.CrankcaseSaturationTemperature.fValue;
   "DB_Application".FromHB.DB_Calc.Compressor_CrankcaseSuperheat               := "DB_Calc".Compressor.CrankcaseSuperheat.fValue;
   "DB_Application".FromHB.DB_Calc.Compressor_VolumetricEfficiency             := "DB_Calc".Compressor.VolumetricEfficiency.fValue;
   "DB_Application".FromHB.DB_Calc.Compressor_IsentropicEfficiency             := "DB_Calc".Compressor.IsentropicEfficiency.fValue;
   "DB_Application".FromHB.DB_Calc.Compressor_Massflow                         := "DB_Calc".Compressor.Massflow.fValue;

   "DB_Application".FromHB.DB_Calc.Heatsink_DeltaT                             := "DB_Calc".HeatSink.DeltaT.fValue;
   "DB_Application".FromHB.DB_Calc.Heatsink_Pinch                              := "DB_Calc".HeatSink.Pinch.fValue;
   "DB_Application".FromHB.DB_Calc.Heatsink_Heatrate                           := "DB_Calc".HeatSink.HeatRate.fValue;
   "DB_Application".FromHB.DB_Calc.Heatsink_DeltaP                             := "DB_Calc".HeatSink.DeltaP.fValue;
   "DB_Application".FromHB.DB_Calc.Heatsink_Massflow                           := "DB_Calc".HeatSink.Massflow.fValue;

   "DB_Application".FromHB.DB_Calc.Heatsource_DeltaT                           := "DB_Calc".HeatSource.DeltaT.fValue;
   "DB_Application".FromHB.DB_Calc.Heatsource_Pinch                            := "DB_Calc".HeatSource.Pinch.fValue;
   "DB_Application".FromHB.DB_Calc.Heatsource_Heatrate                         := "DB_Calc".HeatSource.HeatRate.fValue;
   "DB_Application".FromHB.DB_Calc.Heatsource_DeltaP                           := "DB_Calc".HeatSource.DeltaP.fValue;
   "DB_Application".FromHB.DB_Calc.Heatsource_Massflow                         := "DB_Calc".HeatSource.Massflow.fValue;
   "DB_Application".FromHB.DB_Calc.Heatsource_TemperatureRateOfChange          := "DB_Calc".HeatSource.TemperatureRateOfChange.fValue;

   "DB_Application".FromHB.DB_Calc.HighPressPart_CompressorSaturationTemperature := "DB_Calc".HighPressPart.CompressorSaturationTemperature.fValue;
   "DB_Application".FromHB.DB_Calc.HighPressPart_CompressorSuperheat           := "DB_Calc".HighPressPart.CompressorSuperheat.fValue;
   "DB_Application".FromHB.DB_Calc.HighPressPart_CondenserSaturationTemperature:= "DB_Calc".HighPressPart.CondenserSaturationTemperature.fValue;
   "DB_Application".FromHB.DB_Calc.HighPressPart_CondenserSubcooling           := "DB_Calc".HighPressPart.CondenserSubcooling.fValue;
   "DB_Application".FromHB.DB_Calc.HighPressPart_ExpansionValveSubcooling      := "DB_Calc".HighPressPart.ExpansionValveSubcooling.fValue;
   "DB_Application".FromHB.DB_Calc.HighPressPart_CondenserDeltaP               := "DB_Calc".HighPressPart.CondenserDeltaP.fValue;

   "DB_Application".FromHB.DB_Calc.LowPressPart_EvaporatorSuperheat            := "DB_Calc".LowPressPart.EvaporatorSuperheat.fValue;
   "DB_Application".FromHB.DB_Calc.LowPressPart_CompressorSuperheat            := "DB_Calc".LowPressPart.CompressorSuperheat.fValue;
   "DB_Application".FromHB.DB_Calc.LowPressPart_EvaporatorSaturationTemperature:= "DB_Calc".LowPressPart.EvaporatorSaturationTemperature.fValue;
   "DB_Application".FromHB.DB_Calc.LowPressPart_CompressorSaturationTemperature:= "DB_Calc".LowPressPart.CompressorSaturationTemperature.fValue;

   "DB_Application".FromHB.DB_Calc.System_Quality                              := "DB_Calc".System.Quality.fValue;
   "DB_Application".FromHB.DB_Calc.System_COP                                  := "DB_Calc".System.COP.fValue;
   "DB_Application".FromHB.DB_Calc.System_ElectricalPower                      := "DB_Calc".System.ElectricalPower.fValue;
   "DB_Application".FromHB.DB_Calc.System_TemperatureLift                      := "DB_Calc".System.TemperatureLift.fValue;
   "DB_Application".FromHB.DB_Calc.System_MotorEfficiency                      := "DB_Calc".System.MotorEfficiency.fValue;
   "DB_Application".FromHB.DB_Calc.System_FMEP                                 := "DB_Calc".System.FMEP.fValue;

   "DB_Application".FromHB.DB_Calc.Aux_ShaftSealDeltaT                         := "DB_Calc".Auxiliary.ShaftSealDeltaT.fValue;
   "DB_Application".FromHB.DB_Calc.Aux_CPCPumpDeltaP                           := "DB_Calc".Auxiliary.CPCDeltaP.fValue;

   "DB_Application".FromHB.DB_Calc.Misc_EvaporatorDischargePressureMean        := "DB_Calc".Misc.EvaporatorDischargePressureMean.fValue;
   "DB_Application".FromHB.DB_Calc.Misc_EvaporatorDischargeTemperatureMin      := "DB_Calc".Misc.EvaporatorDischargeTemperatureMin.fValue;
   "DB_Application".FromHB.DB_Calc.Misc_EvaporatorDischargeTemperatureMean     := "DB_Calc".Misc.EvaporatorDischargeTemperatureMean.fValue;
   "DB_Application".FromHB.DB_Calc.Misc_OilFilterDeltaP                        := "DB_Calc".Misc.OilFilterDeltaP.fValue;
END_REGION

REGION Network 4 (SCL): DB_InverterDrives & DB_Valves
   // Done this way for minimum bandwidth
   "DB_Application".FromHB.DB_InverterDrives.HBL_SC_01_A1  := "DB_InverterDrives".HBL_SC_01.Stat.Speed.Eng.fValue;
   "DB_Application".FromHB.DB_InverterDrives.HBL_SC_01_A2  := "DB_InverterDrives".HBL_SC_01.Stat.Torque.Eng.fValue;
   "DB_Application".FromHB.DB_InverterDrives.HBL_SC_01_A3  := "DB_InverterDrives".HBL_SC_01.Stat.Power.Eng.fValue;
   "DB_Application".FromHB.DB_InverterDrives.HBL_SC_02_A1  := "DB_InverterDrives".HBL_SC_02.Stat.Speed.Eng.fValue;
   "DB_Application".FromHB.DB_InverterDrives.HBL_SC_02_A2  := "DB_InverterDrives".HBL_SC_02.Stat.Torque.Eng.fValue;
   "DB_Application".FromHB.DB_InverterDrives.HBL_SC_02_A3  := "DB_InverterDrives".HBL_SC_02.Stat.Power.Eng.fValue;
   "DB_Application".FromHB.DB_InverterDrives.HBL_SC_10_A1  := "DB_InverterDrives".HBL_SC_10.Stat.Speed.Eng.fValue;
   "DB_Application".FromHB.DB_InverterDrives.HBL_SC_10_A2  := "DB_InverterDrives".HBL_SC_10.Stat.Torque.Eng.fValue;
   "DB_Application".FromHB.DB_InverterDrives.HBL_SC_10_A3  := "DB_InverterDrives".HBL_SC_10.Stat.Power.Eng.fValue;
   "DB_Application".FromHB.DB_InverterDrives.HBL_SC_03_A1  := "DB_InverterDrives".HBL_SC_03.Stat.Speed.Eng.fValue;
   "DB_Application".FromHB.DB_InverterDrives.HBL_SC_03_A2  := "DB_InverterDrives".HBL_SC_03.Stat.Torque.Eng.fValue;
   "DB_Application".FromHB.DB_InverterDrives.HBL_SC_03_A3  := "DB_InverterDrives".HBL_SC_03.Stat.Power.Eng.fValue;

   "DB_Application".FromHB.DB_Valves.HBL_HCV_576_A1        := "DB_Valves".HBL_HCV_576.Stat.Position.Eng.fValue;
   "DB_Application".FromHB.DB_Valves.HBL_HCV_577_A1        := "DB_Valves".HBL_HCV_577.Stat.Position.Eng.fValue;
   "DB_Application".FromHB.DB_Valves.HBL_HCV_578_A1        := "DB_Valves".HBL_HCV_578.Stat.Position.Eng.fValue;
   "DB_Application".FromHB.DB_Valves.HBL_HCV_579_A1        := "DB_Valves".HBL_HCV_579.Stat.Position.Eng.fValue;
   "DB_Application".FromHB.DB_Valves.HBL_HCV_515_A1        := "DB_Valves".HBL_HCV_515.Stat.Position.Eng.fValue;
   "DB_Application".FromHB.DB_Valves.HBL_HCV_575_A1        := "DB_Valves".HBL_HCV_575.Stat.Position.Eng.fValue;
   "DB_Application".FromHB.DB_Valves.HBL_HCV_616_A1        := "DB_Valves".HBL_HCV_616.Stat.Position.Eng.fValue;
   "DB_Application".FromHB.DB_Valves.HBL_HCV_700_A1        := "DB_Valves".HBL_HCV_700.Stat.Position.Eng.fValue;
   "DB_Application".FromHB.DB_Valves.HBL_HCV_514_A1        := "DB_Valves".HBL_HCV_514.Stat.Position.Eng.fValue;
   "DB_Application".FromHB.DB_Valves.HBL_HCV_548_A1        := "DB_Valves".HBL_HCV_548.Stat.Position.Eng.fValue;
END_REGION

REGION Network 5 (SCL): Commands
   // Application PLC PUTs these, so no code here :-)
END_REGION

REGION Network 6: Watchdog/liveness bit
   // Check if data is valid from external systems
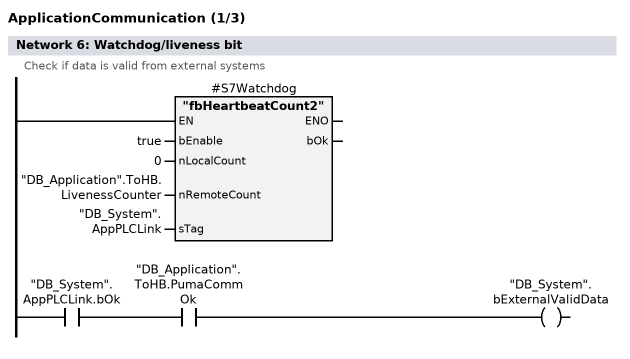
   RUNG wire#powerrail
      #S7Watchdog(bEnable := true, nLocalCount := 0, nRemoteCount := "DB_Application".ToHB.LivenessCounter, sTag := "DB_System".AppPLCLink, bOk =>)
   END_RUNG
   RUNG wire#powerrail
      Contact( "DB_System".AppPLCLink.bOk )
      Contact( "DB_Application".ToHB.PumaCommOk )
      Coil( "DB_System".bExternalValidData )
   END_RUNG
   // the same network as SCL:
   #S7Watchdog(bEnable := true,   // "fbHeartbeatCount2"
               nLocalCount := 0,
               nRemoteCount := "DB_Application".ToHB.LivenessCounter,
               sTag := "DB_System".AppPLCLink);
   "DB_System".bExternalValidData := "DB_System".AppPLCLink.bOk AND "DB_Application".ToHB.PumaCommOk;
END_REGION

REGION Network 7: Process setpoints from Application PLC
   // A positive edge followed by a SET  writes to the destination bit once, without "holding" the value. Easiest to write & read in ladder.
   // Triggering a MOVE on value change writes the value once without continually overwriting it.
   // A negative edge followed by a RESET writes to the destination bit once, without "holding" the value. Easiest to write & read in ladder.
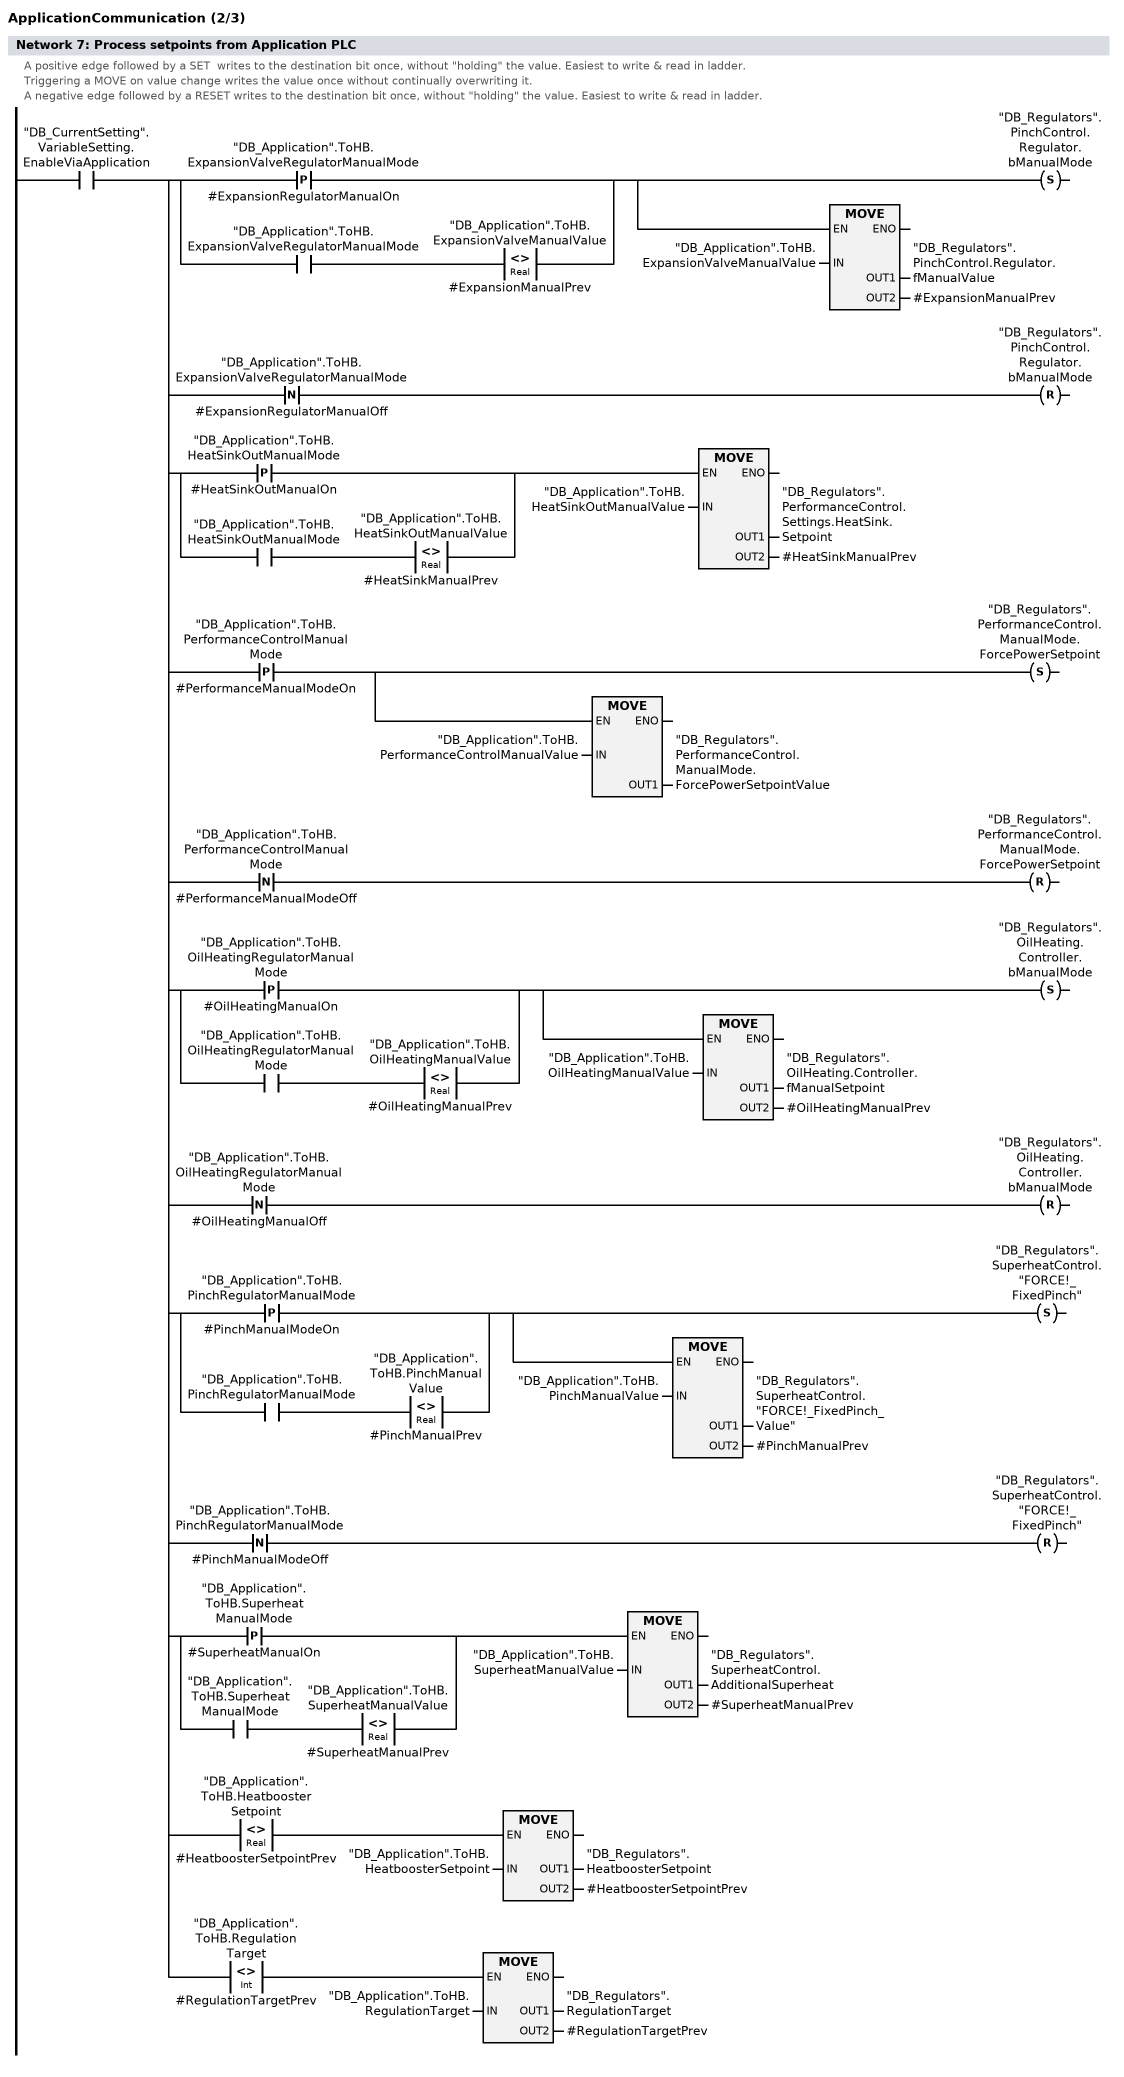
   RUNG wire#powerrail
      Contact( "DB_CurrentSetting".VariableSetting.EnableViaApplication )
      wire#w1
      P_Contact(operand := "DB_Application".ToHB.ExpansionValveRegulatorManualMode, bit := #ExpansionRegulatorManualOn)
      wire#w2
      S_Coil( "DB_Regulators".PinchControl.Regulator.bManualMode )
   END_RUNG
   RUNG wire#w1
      Contact( "DB_Application".ToHB.ExpansionValveRegulatorManualMode )
      { S7_Templates := "SrcType := Real" } NE_Contact(in1 := "DB_Application".ToHB.ExpansionValveManualValue, in2 := #ExpansionManualPrev)
   END_RUNG wire#w2
   RUNG wire#w2
      Move(in := "DB_Application".ToHB.ExpansionValveManualValue, out1 => "DB_Regulators".PinchControl.Regulator.fManualValue, out2 => #ExpansionManualPrev)
   END_RUNG
   RUNG wire#w1
      N_Contact(operand := "DB_Application".ToHB.ExpansionValveRegulatorManualMode, bit := #ExpansionRegulatorManualOff)
      R_Coil( "DB_Regulators".PinchControl.Regulator.bManualMode )
   END_RUNG
   RUNG wire#w1
      P_Contact(operand := "DB_Application".ToHB.HeatSinkOutManualMode, bit := #HeatSinkOutManualOn)
      wire#w3
      Move(in := "DB_Application".ToHB.HeatSinkOutManualValue, out1 => "DB_Regulators".PerformanceControl.Settings.HeatSink.Setpoint, out2 => #HeatSinkManualPrev)
   END_RUNG
   RUNG wire#w1
      Contact( "DB_Application".ToHB.HeatSinkOutManualMode )
      { S7_Templates := "SrcType := Real" } NE_Contact(in1 := "DB_Application".ToHB.HeatSinkOutManualValue, in2 := #HeatSinkManualPrev)
   END_RUNG wire#w3
   RUNG wire#w1
      P_Contact(operand := "DB_Application".ToHB.PerformanceControlManualMode, bit := #PerformanceManualModeOn)
      wire#w4
      S_Coil( "DB_Regulators".PerformanceControl.ManualMode.ForcePowerSetpoint )
   END_RUNG
   RUNG wire#w4
      Move(in := "DB_Application".ToHB.PerformanceControlManualValue, out1 => "DB_Regulators".PerformanceControl.ManualMode.ForcePowerSetpointValue)
   END_RUNG
   RUNG wire#w1
      N_Contact(operand := "DB_Application".ToHB.PerformanceControlManualMode, bit := #PerformanceManualModeOff)
      R_Coil( "DB_Regulators".PerformanceControl.ManualMode.ForcePowerSetpoint )
   END_RUNG
   RUNG wire#w1
      P_Contact(operand := "DB_Application".ToHB.OilHeatingRegulatorManualMode, bit := #OilHeatingManualOn)
      wire#w5
      S_Coil( "DB_Regulators".OilHeating.Controller.bManualMode )
   END_RUNG
   RUNG wire#w1
      Contact( "DB_Application".ToHB.OilHeatingRegulatorManualMode )
      { S7_Templates := "SrcType := Real" } NE_Contact(in1 := "DB_Application".ToHB.OilHeatingManualValue, in2 := #OilHeatingManualPrev)
   END_RUNG wire#w5
   RUNG wire#w5
      Move(in := "DB_Application".ToHB.OilHeatingManualValue, out1 => "DB_Regulators".OilHeating.Controller.fManualSetpoint, out2 => #OilHeatingManualPrev)
   END_RUNG
   RUNG wire#w1
      N_Contact(operand := "DB_Application".ToHB.OilHeatingRegulatorManualMode, bit := #OilHeatingManualOff)
      R_Coil( "DB_Regulators".OilHeating.Controller.bManualMode )
   END_RUNG
   RUNG wire#w1
      P_Contact(operand := "DB_Application".ToHB.PinchRegulatorManualMode, bit := #PinchManualModeOn)
      wire#w6
      S_Coil( "DB_Regulators".SuperheatControl."FORCE!_FixedPinch" )
   END_RUNG
   RUNG wire#w1
      Contact( "DB_Application".ToHB.PinchRegulatorManualMode )
      { S7_Templates := "SrcType := Real" } NE_Contact(in1 := "DB_Application".ToHB.PinchManualValue, in2 := #PinchManualPrev)
   END_RUNG wire#w6
   RUNG wire#w6
      Move(in := "DB_Application".ToHB.PinchManualValue, out1 => "DB_Regulators".SuperheatControl."FORCE!_FixedPinch_Value", out2 => #PinchManualPrev)
   END_RUNG
   RUNG wire#w1
      N_Contact(operand := "DB_Application".ToHB.PinchRegulatorManualMode, bit := #PinchManualModeOff)
      R_Coil( "DB_Regulators".SuperheatControl."FORCE!_FixedPinch" )
   END_RUNG
   RUNG wire#w1
      P_Contact(operand := "DB_Application".ToHB.SuperheatManualMode, bit := #SuperheatManualOn)
      wire#w7
      Move(in := "DB_Application".ToHB.SuperheatManualValue, out1 => "DB_Regulators".SuperheatControl.AdditionalSuperheat, out2 => #SuperheatManualPrev)
   END_RUNG
   RUNG wire#w1
      Contact( "DB_Application".ToHB.SuperheatManualMode )
      { S7_Templates := "SrcType := Real" } NE_Contact(in1 := "DB_Application".ToHB.SuperheatManualValue, in2 := #SuperheatManualPrev)
   END_RUNG wire#w7
   RUNG wire#w1
      { S7_Templates := "SrcType := Real" } NE_Contact(in1 := "DB_Application".ToHB.HeatboosterSetpoint, in2 := #HeatboosterSetpointPrev)
      Move(in := "DB_Application".ToHB.HeatboosterSetpoint, out1 => "DB_Regulators".HeatboosterSetpoint, out2 => #HeatboosterSetpointPrev)
   END_RUNG
   RUNG wire#w1
      { S7_Templates := "SrcType := Int" } NE_Contact(in1 := "DB_Application".ToHB.RegulationTarget, in2 := #RegulationTargetPrev)
      Move(in := "DB_Application".ToHB.RegulationTarget, out1 => "DB_Regulators".RegulationTarget, out2 => #RegulationTargetPrev)
   END_RUNG
   // the same network as SCL:
   #_w1 := "DB_CurrentSetting".VariableSetting.EnableViaApplication AND "DB_Application".ToHB.ExpansionValveRegulatorManualMode AND NOT #ExpansionRegulatorManualOn;   // rising edge of "DB_Application".ToHB.ExpansionValveRegulatorManualMode
   #ExpansionRegulatorManualOn := "DB_Application".ToHB.ExpansionValveRegulatorManualMode;
   IF #_w1 OR ("DB_CurrentSetting".VariableSetting.EnableViaApplication AND "DB_Application".ToHB.ExpansionValveRegulatorManualMode AND ("DB_Application".ToHB.ExpansionValveManualValue <> #ExpansionManualPrev)) THEN
       "DB_Regulators".PinchControl.Regulator.bManualMode := TRUE;
       "DB_Regulators".PinchControl.Regulator.fManualValue := "DB_Application".ToHB.ExpansionValveManualValue;
       #ExpansionManualPrev := "DB_Application".ToHB.ExpansionValveManualValue;
   END_IF;
   #_w2 := "DB_CurrentSetting".VariableSetting.EnableViaApplication AND NOT "DB_Application".ToHB.ExpansionValveRegulatorManualMode AND #ExpansionRegulatorManualOff;   // falling edge of "DB_Application".ToHB.ExpansionValveRegulatorManualMode
   #ExpansionRegulatorManualOff := "DB_Application".ToHB.ExpansionValveRegulatorManualMode;
   IF #_w2 THEN "DB_Regulators".PinchControl.Regulator.bManualMode := FALSE; END_IF;
   #_w3 := "DB_CurrentSetting".VariableSetting.EnableViaApplication AND "DB_Application".ToHB.HeatSinkOutManualMode AND NOT #HeatSinkOutManualOn;   // rising edge of "DB_Application".ToHB.HeatSinkOutManualMode
   #HeatSinkOutManualOn := "DB_Application".ToHB.HeatSinkOutManualMode;
   IF #_w3 OR ("DB_CurrentSetting".VariableSetting.EnableViaApplication AND "DB_Application".ToHB.HeatSinkOutManualMode AND ("DB_Application".ToHB.HeatSinkOutManualValue <> #HeatSinkManualPrev)) THEN
       "DB_Regulators".PerformanceControl.Settings.HeatSink.Setpoint := "DB_Application".ToHB.HeatSinkOutManualValue;
       #HeatSinkManualPrev := "DB_Application".ToHB.HeatSinkOutManualValue;
   END_IF;
   #_w4 := "DB_CurrentSetting".VariableSetting.EnableViaApplication AND "DB_Application".ToHB.PerformanceControlManualMode AND NOT #PerformanceManualModeOn;   // rising edge of "DB_Application".ToHB.PerformanceControlManualMode
   #PerformanceManualModeOn := "DB_Application".ToHB.PerformanceControlManualMode;
   IF #_w4 THEN
       "DB_Regulators".PerformanceControl.ManualMode.ForcePowerSetpoint := TRUE;
       "DB_Regulators".PerformanceControl.ManualMode.ForcePowerSetpointValue := "DB_Application".ToHB.PerformanceControlManualValue;
   END_IF;
   #_w5 := "DB_CurrentSetting".VariableSetting.EnableViaApplication AND NOT "DB_Application".ToHB.PerformanceControlManualMode AND #PerformanceManualModeOff;   // falling edge of "DB_Application".ToHB.PerformanceControlManualMode
   #PerformanceManualModeOff := "DB_Application".ToHB.PerformanceControlManualMode;
   IF #_w5 THEN "DB_Regulators".PerformanceControl.ManualMode.ForcePowerSetpoint := FALSE; END_IF;
   #_w6 := "DB_CurrentSetting".VariableSetting.EnableViaApplication AND "DB_Application".ToHB.OilHeatingRegulatorManualMode AND NOT #OilHeatingManualOn;   // rising edge of "DB_Application".ToHB.OilHeatingRegulatorManualMode
   #OilHeatingManualOn := "DB_Application".ToHB.OilHeatingRegulatorManualMode;
   IF #_w6 OR ("DB_CurrentSetting".VariableSetting.EnableViaApplication AND "DB_Application".ToHB.OilHeatingRegulatorManualMode AND ("DB_Application".ToHB.OilHeatingManualValue <> #OilHeatingManualPrev)) THEN
       "DB_Regulators".OilHeating.Controller.bManualMode := TRUE;
       "DB_Regulators".OilHeating.Controller.fManualSetpoint := "DB_Application".ToHB.OilHeatingManualValue;
       #OilHeatingManualPrev := "DB_Application".ToHB.OilHeatingManualValue;
   END_IF;
   #_w7 := "DB_CurrentSetting".VariableSetting.EnableViaApplication AND NOT "DB_Application".ToHB.OilHeatingRegulatorManualMode AND #OilHeatingManualOff;   // falling edge of "DB_Application".ToHB.OilHeatingRegulatorManualMode
   #OilHeatingManualOff := "DB_Application".ToHB.OilHeatingRegulatorManualMode;
   IF #_w7 THEN "DB_Regulators".OilHeating.Controller.bManualMode := FALSE; END_IF;
   #_w8 := "DB_CurrentSetting".VariableSetting.EnableViaApplication AND "DB_Application".ToHB.PinchRegulatorManualMode AND NOT #PinchManualModeOn;   // rising edge of "DB_Application".ToHB.PinchRegulatorManualMode
   #PinchManualModeOn := "DB_Application".ToHB.PinchRegulatorManualMode;
   IF #_w8 OR ("DB_CurrentSetting".VariableSetting.EnableViaApplication AND "DB_Application".ToHB.PinchRegulatorManualMode AND ("DB_Application".ToHB.PinchManualValue <> #PinchManualPrev)) THEN
       "DB_Regulators".SuperheatControl."FORCE!_FixedPinch" := TRUE;
       "DB_Regulators".SuperheatControl."FORCE!_FixedPinch_Value" := "DB_Application".ToHB.PinchManualValue;
       #PinchManualPrev := "DB_Application".ToHB.PinchManualValue;
   END_IF;
   #_w9 := "DB_CurrentSetting".VariableSetting.EnableViaApplication AND NOT "DB_Application".ToHB.PinchRegulatorManualMode AND #PinchManualModeOff;   // falling edge of "DB_Application".ToHB.PinchRegulatorManualMode
   #PinchManualModeOff := "DB_Application".ToHB.PinchRegulatorManualMode;
   IF #_w9 THEN "DB_Regulators".SuperheatControl."FORCE!_FixedPinch" := FALSE; END_IF;
   #_w10 := "DB_CurrentSetting".VariableSetting.EnableViaApplication AND "DB_Application".ToHB.SuperheatManualMode AND NOT #SuperheatManualOn;   // rising edge of "DB_Application".ToHB.SuperheatManualMode
   #SuperheatManualOn := "DB_Application".ToHB.SuperheatManualMode;
   IF #_w10 OR ("DB_CurrentSetting".VariableSetting.EnableViaApplication AND "DB_Application".ToHB.SuperheatManualMode AND ("DB_Application".ToHB.SuperheatManualValue <> #SuperheatManualPrev)) THEN
       "DB_Regulators".SuperheatControl.AdditionalSuperheat := "DB_Application".ToHB.SuperheatManualValue;
       #SuperheatManualPrev := "DB_Application".ToHB.SuperheatManualValue;
   END_IF;
   IF "DB_CurrentSetting".VariableSetting.EnableViaApplication AND ("DB_Application".ToHB.HeatboosterSetpoint <> #HeatboosterSetpointPrev) THEN
       "DB_Regulators".HeatboosterSetpoint := "DB_Application".ToHB.HeatboosterSetpoint;
       #HeatboosterSetpointPrev := "DB_Application".ToHB.HeatboosterSetpoint;
   END_IF;
   IF "DB_CurrentSetting".VariableSetting.EnableViaApplication AND ("DB_Application".ToHB.RegulationTarget <> #RegulationTargetPrev) THEN
       "DB_Regulators".RegulationTarget := "DB_Application".ToHB.RegulationTarget;
       #RegulationTargetPrev := "DB_Application".ToHB.RegulationTarget;
   END_IF;
END_REGION

REGION Network 8: Process commands from Application PLC
   // Start & stop requests handled by FB30 StartStopControl
   // FastStop handled by FB34 MotorControl
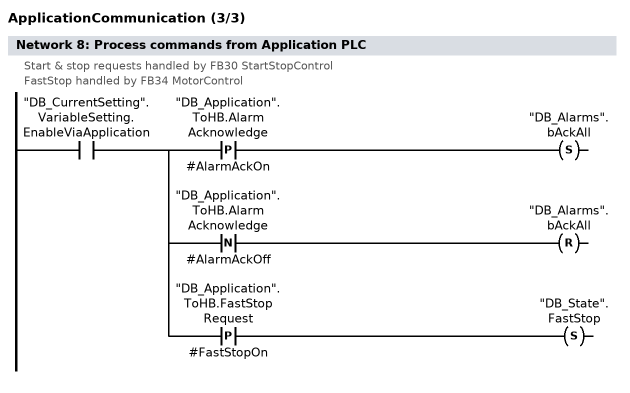
   RUNG wire#powerrail
      Contact( "DB_CurrentSetting".VariableSetting.EnableViaApplication )
      wire#w1
      P_Contact(operand := "DB_Application".ToHB.AlarmAcknowledge, bit := #AlarmAckOn)
      S_Coil( "DB_Alarms".bAckAll )
   END_RUNG
   RUNG wire#w1
      N_Contact(operand := "DB_Application".ToHB.AlarmAcknowledge, bit := #AlarmAckOff)
      R_Coil( "DB_Alarms".bAckAll )
   END_RUNG
   RUNG wire#w1
      P_Contact(operand := "DB_Application".ToHB.FastStopRequest, bit := #FastStopOn)
      S_Coil( "DB_State".FastStop )
   END_RUNG
   // the same network as SCL:
   #_w1 := "DB_CurrentSetting".VariableSetting.EnableViaApplication AND "DB_Application".ToHB.AlarmAcknowledge AND NOT #AlarmAckOn;   // rising edge of "DB_Application".ToHB.AlarmAcknowledge
   #AlarmAckOn := "DB_Application".ToHB.AlarmAcknowledge;
   IF #_w1 THEN "DB_Alarms".bAckAll := TRUE; END_IF;
   #_w2 := "DB_CurrentSetting".VariableSetting.EnableViaApplication AND NOT "DB_Application".ToHB.AlarmAcknowledge AND #AlarmAckOff;   // falling edge of "DB_Application".ToHB.AlarmAcknowledge
   #AlarmAckOff := "DB_Application".ToHB.AlarmAcknowledge;
   IF #_w2 THEN "DB_Alarms".bAckAll := FALSE; END_IF;
   #_w3 := "DB_CurrentSetting".VariableSetting.EnableViaApplication AND "DB_Application".ToHB.FastStopRequest AND NOT #FastStopOn;   // rising edge of "DB_Application".ToHB.FastStopRequest
   #FastStopOn := "DB_Application".ToHB.FastStopRequest;
   IF #_w3 THEN "DB_State".FastStop := TRUE; END_IF;
END_REGION
END_FUNCTION_BLOCK

ORGANIZATION_BLOCK "Time error interrupt"   // OB80, FBD, TimeErrorInterrupt
{ S7_Optimized_Access := 'TRUE' }
VERSION : 0.1
// stored: IsIECCheckEnabled false, SetENOAutomatically false
   VAR_INPUT
      Fault_ID : Byte;   // Fault identifier
      Csg_OBnr : OB_ANY;   // Number of OB causing the error
      Csg_Prio : UInt;   // Priority of OB causing the error
   END_VAR
BEGIN

REGION Network 1: Cycle timeout detection
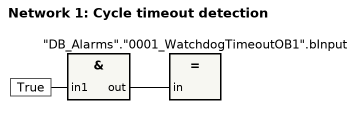
   "DB_Alarms"."0001_WatchdogTimeoutOB1".bInput := True;
END_REGION
END_ORGANIZATION_BLOCK

FUNCTION "SaturationPressure" : Void   // FC28, FBD
{ S7_Optimized_Access := 'TRUE' }
VERSION : 0.1
// stored: AutoNumber true, IsIECCheckEnabled false, SetENOAutomatically false, UDAEnableTagReadback false
   VAR_INPUT
      Temperature : Real;
   END_VAR
   VAR_OUTPUT
      Pressure : Real;
   END_VAR
   VAR_TEMP
      CalcPressure : Real;
   END_VAR
   VAR_TEMP   // added for the SCL form of the ladder/FBD networks
      _w1 : Bool;
   END_VAR
BEGIN

REGION Network 1
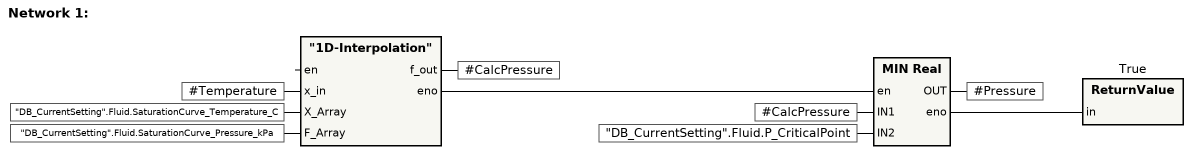
   "1D-Interpolation"(x_in := #Temperature,
                      X_Array := "DB_CurrentSetting".Fluid.SaturationCurve_Temperature_C,
                      F_Array := "DB_CurrentSetting".Fluid.SaturationCurve_Pressure_kPa,
                      f_out => #CalcPressure,
                      ENO => #_w1);
   IF #_w1 THEN
       #Pressure := MIN(IN1 := #CalcPressure, IN2 := "DB_CurrentSetting".Fluid.P_CriticalPoint);
       ENO := True;
       RETURN;
   END_IF;
END_REGION
END_FUNCTION

FUNCTION_BLOCK "fbHoursCounter2"   // FB54, LAD
TITLE = Hours counter
{ S7_Optimized_Access := 'TRUE' }
AUTHOR : Heaten
VERSION : 0.1
// stored: AutoNumber true, IsIECCheckEnabled false, IsRetainMemResEnabled false, MemoryReserve 0, SetENOAutomatically false, UDAEnableTagReadback false
   VAR_INPUT
      bCLK : Bool;   // 1-second pulse
      bEnable : Bool;   // Enable counting
   END_VAR
   VAR_IN_OUT
      sTag : "stHoursCounter";
   END_VAR
   VAR
      Tick : Bool;
      Reset : Bool;
   END_VAR
   VAR_TEMP
      Clock : Bool;
   END_VAR
   VAR_TEMP   // added for the SCL form of the ladder/FBD networks
      _w1 : Bool;
   END_VAR
BEGIN

REGION Network 1: Clock bit
   // When bEnable = TRUE, increase the elapsed time count
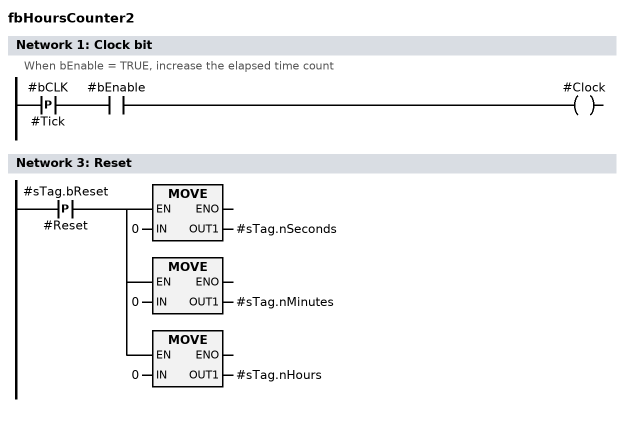
   RUNG wire#powerrail
      P_Contact(operand := #bCLK, bit := #Tick)
      Contact( #bEnable )
      Coil( #Clock )
   END_RUNG
   // the same network as SCL:
   #_w1 := #bCLK AND NOT #Tick;   // rising edge of #bCLK
   #Tick := #bCLK;
   #Clock := #_w1 AND #bEnable;
END_REGION

REGION Network 2 (SCL): Counting
   // Note: this is not automatically reset, should count up "forever" (approx equal to 490293 years).
   IF #Clock = TRUE THEN
       #sTag.nSeconds := #sTag.nSeconds + 1;
       IF #sTag.nSeconds > 59 THEN
           #sTag.nSeconds := 0;
           #sTag.nMinutes := #sTag.nMinutes + 1;
           IF #sTag.nMinutes > 59 THEN
               #sTag.nMinutes := 0;
               #sTag.nHours := #sTag.nHours + 1;
           END_IF;
       END_IF;
   END_IF;
END_REGION

REGION Network 3: Reset
   RUNG wire#powerrail
      P_Contact(operand := #sTag.bReset, bit := #Reset)
      wire#w1
      Move(in := 0, out1 => #sTag.nSeconds)
   END_RUNG
   RUNG wire#w1
      Move(in := 0, out1 => #sTag.nMinutes)
   END_RUNG
   RUNG wire#w1
      Move(in := 0, out1 => #sTag.nHours)
   END_RUNG
   // the same network as SCL:
   #_w1 := #sTag.bReset AND NOT #Reset;   // rising edge of #sTag.bReset
   #Reset := #sTag.bReset;
   IF #_w1 THEN
       #sTag.nSeconds := 0;
       #sTag.nMinutes := 0;
       #sTag.nHours := 0;
   END_IF;
END_REGION
END_FUNCTION_BLOCK

FUNCTION "isNotNaN" : Bool   // FC21, FBD
TITLE = isNotNaN
{ S7_Optimized_Access := 'TRUE' }
VERSION : 0.1
// Returns TRUE if a REAL is not NaN
// stored: AutoNumber true, IsIECCheckEnabled false, SetENOAutomatically false, UDAEnableTagReadback false
   VAR_INPUT
      In : Real;
   END_VAR
BEGIN

REGION Network 1
   // OK is a compiler builtin, but not available in SCL
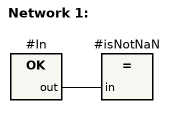
   // no SCL statement known for OK: written as a call
   #isNotNaN := OK(#In);
END_REGION
END_FUNCTION

FUNCTION_BLOCK "fbProcessValve2"
{ S7_Optimized_Access := 'TRUE' }
AUTHOR : Heaten
VERSION : 0.1
   VAR_INPUT 
      bOpenCommand : Bool;   // Command input (do not write directly into sTag)
      bCloseCommand : Bool;   // Command input (do not write directly into sTag)
      bOpenStatus : Bool;   // Status input (do not write directly into sTag)
      bClosedStatus : Bool;   // Status input (do not write directly into sTag)
   END_VAR

   VAR_OUTPUT 
      bOutOpen : Bool;   // Command output
      bOutClose : Bool;   // Command output
      bOpeningError : Bool;   // Alarm output
      bClosingError : Bool;   // Alarm output
   END_VAR

   VAR_IN_OUT 
      sTag : "stProcessValve2";
   END_VAR

   VAR 
      OpenPulse {InstructionName := 'R_TRIG'; LibVersion := '1.0'; S7_SetPoint := 'False'} : R_TRIG;
      ClosePulse {InstructionName := 'R_TRIG'; LibVersion := '1.0'} : R_TRIG;
      OpenTimer {InstructionName := 'TON_TIME'; LibVersion := '1.0'} : TON_TIME;
      CloseTimer {InstructionName := 'TON_TIME'; LibVersion := '1.0'} : TON_TIME;
   END_VAR

   VAR_TEMP 
      bDummy : Bool;
   END_VAR

   VAR CONSTANT 
      UNKNOWN : USInt := 0;
      CLOSED : USInt := 1;
      OPENING : USInt := 2;
      OPEN : USInt := 3;
      CLOSING : USInt := 4;
      CLOSE_ERROR : USInt := 5;
      OPEN_ERROR : USInt := 6;
      NORMALLY_OPEN : Bool := true;
      NORMALLY_CLOSED : Bool := false;
   END_VAR


BEGIN
	// fbProcessValve2 - valve with separate open & close commands and separate open & closed feedback
	// "2" because it has two states, open and closed (not spring return)
	// The state machine runs like the open/closed feedback are limit switches and deactivates the valve drive signal
	
	// Edges to prevent retriggering
	#OpenPulse(CLK := #bOpenCommand);
	#ClosePulse(CLK := #bCloseCommand);
	
	// Timeouts
	#OpenTimer(IN := (#sTag.nState = #OPENING), PT := #sTag.tOpeningTimeout);
	#CloseTimer(IN := (#sTag.nState = #CLOSING), PT := #sTag.tClosingTimeout);
	
	// Copy to tag
	#sTag.bOpenRequest := #bOpenCommand;
	#sTag.bCloseRequest := #bCloseCommand;
	#sTag.bOpenStatus := #bOpenStatus;
	#sTag.bClosedStatus := #bClosedStatus;
	
	// Valve state
	CASE #sTag.nState OF
	    #UNKNOWN : 
	        // Detect state
	        IF #bOpenStatus = TRUE THEN
	            #sTag.nState := #OPEN;
	        ELSIF #bClosedStatus = TRUE THEN
	            #sTag.nState := #CLOSED;
	        ELSE
	            // Neither open nor closed
	            IF #sTag.bNormalState = #NORMALLY_OPEN THEN
	                // Try to open it
	                #sTag.nState := #OPENING;
	                #bOutOpen := TRUE;
	                #bOutClose := FALSE;
	            ELSE
	                // Try to close it
	                #sTag.nState := #CLOSING;
	                #bOutClose := TRUE;
	                #bOutOpen := FALSE;
	            END_IF;
	        END_IF;
	    #CLOSED : 
	        IF #OpenPulse.Q = TRUE THEN
	            #sTag.nState := #OPENING;
	            #bOutOpen := TRUE;
	        END_IF;
	    #OPENING :
	        IF #bOpenStatus = TRUE THEN
	            #sTag.nState := #OPEN;
	            #bOutOpen := FALSE;
	        ELSIF #OpenTimer.Q = TRUE THEN
	            #sTag.nState := #OPEN_ERROR;
	            #bOutOpen := FALSE;
	        END_IF;
	    #OPEN :
	        IF #ClosePulse.Q = TRUE THEN
	            #sTag.nState := #CLOSING;
	            #bOutClose := TRUE;
	        END_IF;
	    #CLOSING : 
	        IF #bClosedStatus = TRUE THEN
	            #sTag.nState := #CLOSED;
	            #bOutClose := FALSE;
	        ELSIF #CloseTimer.Q = TRUE THEN
	            #sTag.nState := #CLOSE_ERROR;
	            #bOutClose := FALSE;
	        END_IF;
	    #CLOSE_ERROR :
	        IF #bClosedStatus = TRUE THEN
	            #sTag.nState := #CLOSED;
	        ELSIF #bOpenCommand = TRUE THEN
	            #sTag.nState := #OPENING;
	        END_IF;
	    #OPEN_ERROR :
	        IF #bOpenStatus = TRUE THEN
	            #sTag.nState := #OPEN;
	        ELSIF #bCloseCommand = TRUE THEN
	            #sTag.nState := #CLOSING;
	        END_IF;
	END_CASE;
	
	
	    
END_FUNCTION_BLOCK

FUNCTION_BLOCK "fbOnOffRegulator3"
{ S7_Optimized_Access := 'TRUE' }
VERSION : 0.1
   VAR_INPUT 
      bEnable : Bool;   // Enable from process. 1 = enabled, 0 = disabled
      bLow : Bool;   // Lower level switch (1 = level is above switch, 0 = level is below switch)
      bHigh : Bool;   // Higher level switch (1 = level is above switch, 0 = level is below switch)
      bAbove : Bool;   // 1 = regulate when above threshold, 0 = regulate when below threshold
      bReset : Bool;   // 1 = reset manual modes
   END_VAR

   VAR_OUTPUT 
      bOutput : Bool;
      bAtSetpoint : Bool;
   END_VAR

   VAR_IN_OUT 
      sTag : "stOnOffRegulator3";
   END_VAR

   VAR 
      ActivationTimer {InstructionName := 'TP_TIME'; LibVersion := '1.0'} : TP_TIME;
   END_VAR

   VAR_TEMP 
      fSetpoint : Real;
      Enabled : Bool;
   END_VAR


BEGIN
	// 1-sided on/off controller with switch trigger and activation timer
	// Output is triggered by a bool input (eg high level switch) and continues running for a set time period. There is no second level switch.
	// Above = 1: regulate when Process Value (PV) above threshold. Eg. cooling, emptying, depressurizing
	// Above = 0: regulate when PV below threshold. Eg. heating, filling, pressurizing
	
	// Reset manual modes.
	IF #bReset THEN
	    #sTag.bManualOverride := FALSE;
	    #sTag.bOverrideCmd := FALSE;
	END_IF;
	
	IF #sTag.bManualOverride = TRUE THEN
	    // In manual override, everything is awesome
	    #sTag.bFault := FALSE;
	    #sTag.bOutput := #sTag.bOverrideCmd;
	    #sTag.bAtSetpoint := NOT(#sTag.bOutput);
	ELSE
	
	    // Enabled when enabled from process and from HMI (Auto)
	    #Enabled := (#bEnable AND #sTag.bEnable);
	
	    // Run controller
	    #ActivationTimer(IN := (#bHigh AND #bAbove) OR (#bLow AND NOT #bAbove),PT := #sTag.nActivationTime, Q => #sTag.bOutput);
	
	    // At setpoint
	    IF #Enabled = TRUE THEN
	        #sTag.bAtSetpoint := NOT(#sTag.bOutput);
	    ELSE
	        #sTag.bAtSetpoint := FALSE;
	    END_IF;
	
	    // Controller fault
	    #sTag.bFault := FALSE;
	
	END_IF;
	
	// Mode
	IF #sTag.bManualOverride = TRUE THEN
	    #sTag.nMode := 3;
	ELSIF #sTag.bEnable = TRUE THEN
	    #sTag.nMode := 1;
	ELSE
	    #sTag.nMode := 0;
	END_IF;
	
	// Local outputs
	#bOutput := #sTag.bOutput;
	#bAtSetpoint := #sTag.bAtSetpoint;
	
	
END_FUNCTION_BLOCK

FUNCTION "Restriction" : Void
{ S7_Optimized_Access := 'TRUE' }
VERSION : 0.1
   VAR_INPUT 
      ID : Int;
      Target : Real;
      Value : Real;
      Kp : Real;
      Tn : Int;
      Tv : Int;
      fCycleTime : Real;
   END_VAR

   VAR_IN_OUT 
      IO : Struct
         ID : Int;
         Error : Real;
         Targed : Real;
         CurrentValue : Real;
         Kp : Real;
         Tn : Int;
         Tv : Int;
      END_STRUCT;
      DT1_storage : Real;
   END_VAR

   VAR_TEMP 
      Error_calc : Real;
   END_VAR


BEGIN
	    #Error_calc := (#Target - #Value)*#Kp - #Tv * "DT1"(u:= #Value*#Kp,T1:=7, fCycleTime:= #fCycleTime, xh_merk:=#DT1_storage);
	            
	    IF #Error_calc < #IO.Error THEN 
	        #IO.ID:=#ID;
	        #IO.Error := #Error_calc;
	        #IO.Kp := #Kp;
	        #IO.Tn := #Tn;
	        #IO.Targed := #Target;
	        #IO.CurrentValue := #Value;
	    END_IF;
END_FUNCTION

FUNCTION "RecTarget" : Real
{ S7_Optimized_Access := 'TRUE' }
VERSION : 0.1
   VAR_INPUT 
      LoadCappacity : Real;
   END_VAR


BEGIN
	//The optimum superheat after the recuperator is between condensate temperature and evaporator outlet temperature. The factor "LoadCappacity" is used to determine where the target temperature should lie in between. If the temperature on the condensate outlet is lower than the Evaporator outlet temperature, the recuperator would work reversely so we added an exception for this case here. 
	//#RecTarged := #LoadCappacity * (MAX(IN1:="DB_SensorInputs".HighPressPart.T_CondensingTemperature-5.0,IN2:="DB_SensorInputs".LowPressPart.T_EvaporationTemperature) - "DB_SensorInputs".LowPressPart.T12_EvaporatorOut); // Alte version bis 04.09.2018 (Problematisch beim Start und wenig Lift; Auch schlechteres Einregelverhalten)
	#RecTarget := #LoadCappacity * (MAX(IN1 := "DB_AI".HBL_TT_611.Eng.fValue, IN2 := "DB_AI".HBL_TT_543.Eng.fValue) - "DB_Calc".LowPressPart.EvaporatorSaturationTemperature.fValue);         // Neue Version ab  04.09.2018
	//#RecTarged := #LoadCappacity * (MAX(IN1 := "DB_SensorInputs".HighPressPart.T06_CondenserOut, IN2 := "DB_SensorInputs".HeatSource."T13_Inlet_(feed)") - "DB_SensorInputs".LowPressPart.T_EvaporationTemperature);        // Alternative Version zu Variante 2. Stabiler gegen Schwingungen, aber möglicherweise dafür konvervativer im Einregelverhalten
END_FUNCTION

FUNCTION "VapPerformance" : Real
{ S7_Optimized_Access := 'TRUE' }
VERSION : 0.1
   VAR_INPUT 
      AddSuperheat : Real;
      Pinch : Real;
   END_VAR

   VAR_TEMP 
      VapPerformance1 : Real;
      VapPerformance2 : Real;
      VapPerformance3 : Real;
   END_VAR


BEGIN
	//The VapOccupRat is an indicator for the occupancy of the evaporator. The pinch on the steam side is compared to the pinch on the liquid side of the evaporator. The Pinch on the liquid side should be smaller by a factor of "Adjust" to demand a balanced performance.
	#VapPerformance1 := 0.7 * (("DB_AI".HBL_TT_546.Eng.fValue - "DB_AI".HBL_TT_543.Eng.fValue) - 2.5 * #Pinch);
	    // This might react better on a huge variation of heat flow mass flows
	    //#VapPerformance := ("DB_SensorInputs".HeatSource."T13_Inlet_(feed)" - "DB_SensorInputs".LowPressPart.T12_EvaporatorOut) - 0.9 * ("DB_SensorInputs".HeatSource."T13_Inlet_(feed)" - "DB_SensorInputs".LowPressPart.T_EvaporationTemperature);
	#VapPerformance2 := - 3*("DB_Calc".LowPressPart.EvaporatorSuperheat.fValue - 0.12 * ("DB_AI".HBL_TT_546.Eng.fValue-"DB_Calc".LowPressPart.EvaporatorSaturationTemperature.fValue));
	
	
	#VapPerformance3 := 1.0 *(#AddSuperheat-"DB_Calc".LowPressPart.EvaporatorSuperheat.fValue + 0.05 * ("DB_AI".HBL_TT_546.Eng.fValue - "DB_AI".HBL_TT_542.Eng.fValue) + (0.1) * #Pinch);
	
	#VapPerformance := #VapPerformance3;
END_FUNCTION

DATA_BLOCK "DB_CurrentSetting"   // DB21
{ S7_Optimized_Access := 'TRUE' }
AUTHOR : AZ
VERSION : 0.1
// stored: AutoNumber true, DBAccessibleFromOPCUA true, DBAccessibleFromWebserver true, InstanceOfName CurrentSetting-STRUCT, InstanceOfType UDT, IsOnlyStoredInLoadMemory false, IsWriteProtectedInAS false
"CurrentSetting-STRUCT"
BEGIN
   Fluid."Name" := 'R1233zdE';
   Fluid.FluidTypeNumber := 2;
   Fluid.SaturationCurve_Temperature_C[0] := -10.0;
   Fluid.SaturationCurve_Temperature_C[1] := -5.4872;
   Fluid.SaturationCurve_Temperature_C[2] := -0.9744;
   Fluid.SaturationCurve_Temperature_C[3] := 3.5385;
   Fluid.SaturationCurve_Temperature_C[4] := 8.0513;
   Fluid.SaturationCurve_Temperature_C[5] := 12.5641;
   Fluid.SaturationCurve_Temperature_C[6] := 17.0769;
   Fluid.SaturationCurve_Temperature_C[7] := 21.5897;
   Fluid.SaturationCurve_Temperature_C[8] := 26.1026;
   Fluid.SaturationCurve_Temperature_C[9] := 30.6154;
   Fluid.SaturationCurve_Temperature_C[10] := 35.1282;
   Fluid.SaturationCurve_Temperature_C[11] := 39.641;
   Fluid.SaturationCurve_Temperature_C[12] := 44.1538;
   Fluid.SaturationCurve_Temperature_C[13] := 48.6667;
   Fluid.SaturationCurve_Temperature_C[14] := 53.1795;
   Fluid.SaturationCurve_Temperature_C[15] := 57.6923;
   Fluid.SaturationCurve_Temperature_C[16] := 62.2051;
   Fluid.SaturationCurve_Temperature_C[17] := 66.7179;
   Fluid.SaturationCurve_Temperature_C[18] := 71.2308;
   Fluid.SaturationCurve_Temperature_C[19] := 75.7436;
   Fluid.SaturationCurve_Temperature_C[20] := 80.2564;
   Fluid.SaturationCurve_Temperature_C[21] := 84.7692;
   Fluid.SaturationCurve_Temperature_C[22] := 89.2821;
   Fluid.SaturationCurve_Temperature_C[23] := 93.7949;
   Fluid.SaturationCurve_Temperature_C[24] := 98.3077;
   Fluid.SaturationCurve_Temperature_C[25] := 102.8205;
   Fluid.SaturationCurve_Temperature_C[26] := 107.3333;
   Fluid.SaturationCurve_Temperature_C[27] := 111.8462;
   Fluid.SaturationCurve_Temperature_C[28] := 116.359;
   Fluid.SaturationCurve_Temperature_C[29] := 120.8718;
   Fluid.SaturationCurve_Temperature_C[30] := 125.3846;
   Fluid.SaturationCurve_Temperature_C[31] := 129.8974;
   Fluid.SaturationCurve_Temperature_C[32] := 134.4103;
   Fluid.SaturationCurve_Temperature_C[33] := 138.9231;
   Fluid.SaturationCurve_Temperature_C[34] := 143.4359;
   Fluid.SaturationCurve_Temperature_C[35] := 147.9487;
   Fluid.SaturationCurve_Temperature_C[36] := 152.4615;
   Fluid.SaturationCurve_Temperature_C[37] := 156.9744;
   Fluid.SaturationCurve_Temperature_C[38] := 161.4872;
   Fluid.SaturationCurve_Temperature_C[39] := 166.0;
   Fluid.SaturationCurve_Temperature_C[40] := 172.9092;
   Fluid.SaturationCurve_Pressure_kPa[0] := 30.3567;
   Fluid.SaturationCurve_Pressure_kPa[1] := 37.5596;
   Fluid.SaturationCurve_Pressure_kPa[2] := 46.0817;
   Fluid.SaturationCurve_Pressure_kPa[3] := 56.0903;
   Fluid.SaturationCurve_Pressure_kPa[4] := 67.7633;
   Fluid.SaturationCurve_Pressure_kPa[5] := 81.2888;
   Fluid.SaturationCurve_Pressure_kPa[6] := 96.865;
   Fluid.SaturationCurve_Pressure_kPa[7] := 114.6997;
   Fluid.SaturationCurve_Pressure_kPa[8] := 135.0095;
   Fluid.SaturationCurve_Pressure_kPa[9] := 158.0203;
   Fluid.SaturationCurve_Pressure_kPa[10] := 183.9659;
   Fluid.SaturationCurve_Pressure_kPa[11] := 213.0886;
   Fluid.SaturationCurve_Pressure_kPa[12] := 245.6381;
   Fluid.SaturationCurve_Pressure_kPa[13] := 281.8717;
   Fluid.SaturationCurve_Pressure_kPa[14] := 322.0539;
   Fluid.SaturationCurve_Pressure_kPa[15] := 366.4563;
   Fluid.SaturationCurve_Pressure_kPa[16] := 415.3576;
   Fluid.SaturationCurve_Pressure_kPa[17] := 469.0435;
   Fluid.SaturationCurve_Pressure_kPa[18] := 527.8071;
   Fluid.SaturationCurve_Pressure_kPa[19] := 591.9489;
   Fluid.SaturationCurve_Pressure_kPa[20] := 661.7775;
   Fluid.SaturationCurve_Pressure_kPa[21] := 737.6098;
   Fluid.SaturationCurve_Pressure_kPa[22] := 819.7723;
   Fluid.SaturationCurve_Pressure_kPa[23] := 908.6015;
   Fluid.SaturationCurve_Pressure_kPa[24] := 1004.446;
   Fluid.SaturationCurve_Pressure_kPa[25] := 1107.666;
   Fluid.SaturationCurve_Pressure_kPa[26] := 1218.639;
   Fluid.SaturationCurve_Pressure_kPa[27] := 1337.757;
   Fluid.SaturationCurve_Pressure_kPa[28] := 1465.436;
   Fluid.SaturationCurve_Pressure_kPa[29] := 1602.111;
   Fluid.SaturationCurve_Pressure_kPa[30] := 1748.251;
   Fluid.SaturationCurve_Pressure_kPa[31] := 1904.356;
   Fluid.SaturationCurve_Pressure_kPa[32] := 2070.969;
   Fluid.SaturationCurve_Pressure_kPa[33] := 2248.688;
   Fluid.SaturationCurve_Pressure_kPa[34] := 2438.177;
   Fluid.SaturationCurve_Pressure_kPa[35] := 2640.193;
   Fluid.SaturationCurve_Pressure_kPa[36] := 2855.623;
   Fluid.SaturationCurve_Pressure_kPa[37] := 3085.555;
   Fluid.SaturationCurve_Pressure_kPa[38] := 3331.466;
   Fluid.SaturationCurve_Pressure_kPa[39] := 3595.998;
   Fluid.SaturationCurve_Pressure_kPa[40] := 4001.0;
   Fluid.DensityCurve_Pressure_kPa[0] := 50.0;
   Fluid.DensityCurve_Pressure_kPa[1] := 74.7475;
   Fluid.DensityCurve_Pressure_kPa[2] := 173.05;
   Fluid.DensityCurve_Pressure_kPa[3] := 388.0866;
   Fluid.DensityCurve_Pressure_kPa[4] := 746.4811;
   Fluid.DensityCurve_Pressure_kPa[5] := 1244.251;
   Fluid.DensityCurve_Pressure_kPa[6] := 1836.598;
   Fluid.DensityCurve_Pressure_kPa[7] := 2441.284;
   Fluid.DensityCurve_Pressure_kPa[8] := 2962.33;
   Fluid.DensityCurve_Pressure_kPa[9] := 3328.69;
   Fluid.DensityCurve_Pressure_kPa[10] := 3526.57;
   Fluid.DensityCurve_Pressure_kPa[11] := 3613.637;
   Fluid.DensityCurve_Pressure_kPa[12] := 4001.0;
   Fluid.DensityCurveLiquide_Densety_kg_m3[0] := 1319.278;
   Fluid.DensityCurveLiquide_Densety_kg_m3[1] := 1297.254;
   Fluid.DensityCurveLiquide_Densety_kg_m3[2] := 1242.459;
   Fluid.DensityCurveLiquide_Densety_kg_m3[3] := 1173.489;
   Fluid.DensityCurveLiquide_Densety_kg_m3[4] := 1098.545;
   Fluid.DensityCurveLiquide_Densety_kg_m3[5] := 1019.4;
   Fluid.DensityCurveLiquide_Densety_kg_m3[6] := 936.68;
   Fluid.DensityCurveLiquide_Densety_kg_m3[7] := 851.4562;
   Fluid.DensityCurveLiquide_Densety_kg_m3[8] := 765.7374;
   Fluid.DensityCurveLiquide_Densety_kg_m3[9] := 682.3312;
   Fluid.DensityCurveLiquide_Densety_kg_m3[10] := 605.4245;
   Fluid.DensityCurveLiquide_Densety_kg_m3[11] := 523.5075;
   Fluid.DensityCurveLiquide_Densety_kg_m3[12] := 455.9911;
   Fluid.DensityCurveVapor_Densety_kg_m3[0] := 2.9405;
   Fluid.DensityCurveVapor_Densety_kg_m3[1] := 4.2862;
   Fluid.DensityCurveVapor_Densety_kg_m3[2] := 9.4624;
   Fluid.DensityCurveVapor_Densety_kg_m3[3] := 20.5809;
   Fluid.DensityCurveVapor_Densety_kg_m3[4] := 39.5976;
   Fluid.DensityCurveVapor_Densety_kg_m3[5] := 68.316;
   Fluid.DensityCurveVapor_Densety_kg_m3[6] := 108.1358;
   Fluid.DensityCurveVapor_Densety_kg_m3[7] := 159.5525;
   Fluid.DensityCurveVapor_Densety_kg_m3[8] := 221.352;
   Fluid.DensityCurveVapor_Densety_kg_m3[9] := 289.9457;
   Fluid.DensityCurveVapor_Densety_kg_m3[10] := 359.0497;
   Fluid.DensityCurveVapor_Densety_kg_m3[11] := 437.3655;
   Fluid.DensityCurveVapor_Densety_kg_m3[12] := 455.9911;
   Fluid.DensityCurveVapor_SuperheatCorrection_a := 0.0;
   Fluid.DensityCurveVapor_SuperheatCorrection_b := 0.0002;
   Fluid.EnthalpyMap_Superheat_C[0] := -20.0;
   Fluid.EnthalpyMap_Superheat_C[1] := -6.0;
   Fluid.EnthalpyMap_Superheat_C[2] := -2.0;
   Fluid.EnthalpyMap_Superheat_C[3] := -0.01;
   Fluid.EnthalpyMap_Superheat_C[4] := 0.01;
   Fluid.EnthalpyMap_Superheat_C[5] := 2.0;
   Fluid.EnthalpyMap_Superheat_C[6] := 6.0;
   Fluid.EnthalpyMap_Superheat_C[7] := 18.0;
   Fluid.EnthalpyMap_Superheat_C[8] := 40.0;
   Fluid.EnthalpyMap_Pressure_kPa[0] := 100.0;
   Fluid.EnthalpyMap_Pressure_kPa[1] := 127.0833;
   Fluid.EnthalpyMap_Pressure_kPa[2] := 234.6644;
   Fluid.EnthalpyMap_Pressure_kPa[3] := 469.9978;
   Fluid.EnthalpyMap_Pressure_kPa[4] := 862.2203;
   Fluid.EnthalpyMap_Pressure_kPa[5] := 1406.974;
   Fluid.EnthalpyMap_Pressure_kPa[6] := 2055.23;
   Fluid.EnthalpyMap_Pressure_kPa[7] := 2716.992;
   Fluid.EnthalpyMap_Pressure_kPa[8] := 3287.218;
   Fluid.EnthalpyMap_Pressure_kPa[9] := 3688.158;
   Fluid.EnthalpyMap_Pressure_kPa[10] := 3904.715;
   Fluid.EnthalpyMap_Pressure_kPa[11] := 4000.0;
   Fluid.EnthalpyMap_Enthalpy_kJ_kg[0,0] := 197.5698;
   Fluid.EnthalpyMap_Enthalpy_kJ_kg[0,1] := 214.1515;
   Fluid.EnthalpyMap_Enthalpy_kJ_kg[0,2] := 218.9438;
   Fluid.EnthalpyMap_Enthalpy_kJ_kg[0,3] := 221.3373;
   Fluid.EnthalpyMap_Enthalpy_kJ_kg[0,4] := 416.1527;
   Fluid.EnthalpyMap_Enthalpy_kJ_kg[0,5] := 417.767;
   Fluid.EnthalpyMap_Enthalpy_kJ_kg[0,6] := 421.028;
   Fluid.EnthalpyMap_Enthalpy_kJ_kg[0,7] := 430.9391;
   Fluid.EnthalpyMap_Enthalpy_kJ_kg[0,8] := 449.5907;
   Fluid.EnthalpyMap_Enthalpy_kJ_kg[1,0] := 205.2355;
   Fluid.EnthalpyMap_Enthalpy_kJ_kg[1,1] := 221.9542;
   Fluid.EnthalpyMap_Enthalpy_kJ_kg[1,2] := 226.7875;
   Fluid.EnthalpyMap_Enthalpy_kJ_kg[1,3] := 229.2018;
   Fluid.EnthalpyMap_Enthalpy_kJ_kg[1,4] := 420.6821;
   Fluid.EnthalpyMap_Enthalpy_kJ_kg[1,5] := 422.3276;
   Fluid.EnthalpyMap_Enthalpy_kJ_kg[1,6] := 425.6502;
   Fluid.EnthalpyMap_Enthalpy_kJ_kg[1,7] := 435.7365;
   Fluid.EnthalpyMap_Enthalpy_kJ_kg[1,8] := 454.6786;
   Fluid.EnthalpyMap_Enthalpy_kJ_kg[2,0] := 227.161;
   Fluid.EnthalpyMap_Enthalpy_kJ_kg[2,1] := 244.2909;
   Fluid.EnthalpyMap_Enthalpy_kJ_kg[2,2] := 249.2492;
   Fluid.EnthalpyMap_Enthalpy_kJ_kg[2,3] := 251.7272;
   Fluid.EnthalpyMap_Enthalpy_kJ_kg[2,4] := 433.2917;
   Fluid.EnthalpyMap_Enthalpy_kJ_kg[2,5] := 435.0327;
   Fluid.EnthalpyMap_Enthalpy_kJ_kg[2,6] := 438.5429;
   Fluid.EnthalpyMap_Enthalpy_kJ_kg[2,7] := 449.1592;
   Fluid.EnthalpyMap_Enthalpy_kJ_kg[2,8] := 468.9681;
   Fluid.EnthalpyMap_Enthalpy_kJ_kg[3,0] := 256.9384;
   Fluid.EnthalpyMap_Enthalpy_kJ_kg[3,1] := 274.7034;
   Fluid.EnthalpyMap_Enthalpy_kJ_kg[3,2] := 279.8614;
   Fluid.EnthalpyMap_Enthalpy_kJ_kg[3,3] := 282.4424;
   Fluid.EnthalpyMap_Enthalpy_kJ_kg[3,4] := 449.3674;
   Fluid.EnthalpyMap_Enthalpy_kJ_kg[3,5] := 451.2598;
   Fluid.EnthalpyMap_Enthalpy_kJ_kg[3,6] := 455.0643;
   Fluid.EnthalpyMap_Enthalpy_kJ_kg[3,7] := 466.4958;
   Fluid.EnthalpyMap_Enthalpy_kJ_kg[3,8] := 487.595;
   Fluid.EnthalpyMap_Enthalpy_kJ_kg[4,0] := 288.6115;
   Fluid.EnthalpyMap_Enthalpy_kJ_kg[4,1] := 307.2277;
   Fluid.EnthalpyMap_Enthalpy_kJ_kg[4,2] := 312.6681;
   Fluid.EnthalpyMap_Enthalpy_kJ_kg[4,3] := 315.398;
   Fluid.EnthalpyMap_Enthalpy_kJ_kg[4,4] := 464.6608;
   Fluid.EnthalpyMap_Enthalpy_kJ_kg[4,5] := 466.762;
   Fluid.EnthalpyMap_Enthalpy_kJ_kg[4,6] := 470.9658;
   Fluid.EnthalpyMap_Enthalpy_kJ_kg[4,7] := 483.4603;
   Fluid.EnthalpyMap_Enthalpy_kJ_kg[4,8] := 506.1447;
   Fluid.EnthalpyMap_Enthalpy_kJ_kg[5,0] := 319.2484;
   Fluid.EnthalpyMap_Enthalpy_kJ_kg[5,1] := 339.0134;
   Fluid.EnthalpyMap_Enthalpy_kJ_kg[5,2] := 344.8686;
   Fluid.EnthalpyMap_Enthalpy_kJ_kg[5,3] := 347.8254;
   Fluid.EnthalpyMap_Enthalpy_kJ_kg[5,4] := 476.8875;
   Fluid.EnthalpyMap_Enthalpy_kJ_kg[5,5] := 479.2968;
   Fluid.EnthalpyMap_Enthalpy_kJ_kg[5,6] := 484.0675;
   Fluid.EnthalpyMap_Enthalpy_kJ_kg[5,7] := 497.9603;
   Fluid.EnthalpyMap_Enthalpy_kJ_kg[5,8] := 522.524;
   Fluid.EnthalpyMap_Enthalpy_kJ_kg[6,0] := 346.9259;
   Fluid.EnthalpyMap_Enthalpy_kJ_kg[6,1] := 368.272;
   Fluid.EnthalpyMap_Enthalpy_kJ_kg[6,2] := 374.7868;
   Fluid.EnthalpyMap_Enthalpy_kJ_kg[6,3] := 378.132;
   Fluid.EnthalpyMap_Enthalpy_kJ_kg[6,4] := 484.4899;
   Fluid.EnthalpyMap_Enthalpy_kJ_kg[6,5] := 487.4372;
   Fluid.EnthalpyMap_Enthalpy_kJ_kg[6,6] := 493.119;
   Fluid.EnthalpyMap_Enthalpy_kJ_kg[6,7] := 508.9522;
   Fluid.EnthalpyMap_Enthalpy_kJ_kg[6,8] := 535.7144;
   Fluid.EnthalpyMap_Enthalpy_kJ_kg[7,0] := 369.9632;
   Fluid.EnthalpyMap_Enthalpy_kJ_kg[7,1] := 393.4236;
   Fluid.EnthalpyMap_Enthalpy_kJ_kg[7,2] := 401.0829;
   Fluid.EnthalpyMap_Enthalpy_kJ_kg[7,3] := 405.235;
   Fluid.EnthalpyMap_Enthalpy_kJ_kg[7,4] := 486.2374;
   Fluid.EnthalpyMap_Enthalpy_kJ_kg[7,5] := 490.3629;
   Fluid.EnthalpyMap_Enthalpy_kJ_kg[7,6] := 497.6848;
   Fluid.EnthalpyMap_Enthalpy_kJ_kg[7,7] := 516.2058;
   Fluid.EnthalpyMap_Enthalpy_kJ_kg[7,8] := 545.3667;
   Fluid.EnthalpyMap_Enthalpy_kJ_kg[8,0] := 387.0381;
   Fluid.EnthalpyMap_Enthalpy_kJ_kg[8,1] := 412.9451;
   Fluid.EnthalpyMap_Enthalpy_kJ_kg[8,2] := 422.6469;
   Fluid.EnthalpyMap_Enthalpy_kJ_kg[8,3] := 429.1883;
   Fluid.EnthalpyMap_Enthalpy_kJ_kg[8,4] := 480.7851;
   Fluid.EnthalpyMap_Enthalpy_kJ_kg[8,5] := 488.3624;
   Fluid.EnthalpyMap_Enthalpy_kJ_kg[8,6] := 498.5881;
   Fluid.EnthalpyMap_Enthalpy_kJ_kg[8,7] := 520.3678;
   Fluid.EnthalpyMap_Enthalpy_kJ_kg[8,8] := 551.7377;
   Fluid.EnthalpyMap_Enthalpy_kJ_kg[9,0] := 397.8677;
   Fluid.EnthalpyMap_Enthalpy_kJ_kg[9,1] := 425.8558;
   Fluid.EnthalpyMap_Enthalpy_kJ_kg[9,2] := 438.3909;
   Fluid.EnthalpyMap_Enthalpy_kJ_kg[9,3] := 462.7447;
   Fluid.EnthalpyMap_Enthalpy_kJ_kg[9,4] := 463.5576;
   Fluid.EnthalpyMap_Enthalpy_kJ_kg[9,5] := 484.1742;
   Fluid.EnthalpyMap_Enthalpy_kJ_kg[9,6] := 497.9508;
   Fluid.EnthalpyMap_Enthalpy_kJ_kg[9,7] := 522.3931;
   Fluid.EnthalpyMap_Enthalpy_kJ_kg[9,8] := 555.3659;
   Fluid.EnthalpyMap_Enthalpy_kJ_kg[10,0] := 403.7939;
   Fluid.EnthalpyMap_Enthalpy_kJ_kg[10,1] := 433.1682;
   Fluid.EnthalpyMap_Enthalpy_kJ_kg[10,2] := 448.1372;
   Fluid.EnthalpyMap_Enthalpy_kJ_kg[10,3] := 467.0842;
   Fluid.EnthalpyMap_Enthalpy_kJ_kg[10,4] := 467.3177;
   Fluid.EnthalpyMap_Enthalpy_kJ_kg[10,5] := 483.0886;
   Fluid.EnthalpyMap_Enthalpy_kJ_kg[10,6] := 498.0977;
   Fluid.EnthalpyMap_Enthalpy_kJ_kg[10,7] := 523.751;
   Fluid.EnthalpyMap_Enthalpy_kJ_kg[10,8] := 557.4834;
   Fluid.EnthalpyMap_Enthalpy_kJ_kg[11,0] := 406.426;
   Fluid.EnthalpyMap_Enthalpy_kJ_kg[11,1] := 436.4671;
   Fluid.EnthalpyMap_Enthalpy_kJ_kg[11,2] := 452.4549;
   Fluid.EnthalpyMap_Enthalpy_kJ_kg[11,3] := 469.0933;
   Fluid.EnthalpyMap_Enthalpy_kJ_kg[11,4] := 469.2745;
   Fluid.EnthalpyMap_Enthalpy_kJ_kg[11,5] := 483.1994;
   Fluid.EnthalpyMap_Enthalpy_kJ_kg[11,6] := 498.3468;
   Fluid.EnthalpyMap_Enthalpy_kJ_kg[11,7] := 524.4174;
   Fluid.EnthalpyMap_Enthalpy_kJ_kg[11,8] := 558.4523;
   Fluid.Limits.T_HeatSourceTemperature_Max := 120.0;
   Fluid.Limits.T_HeatSourceTemperature_Min := 55.0;
   Fluid.Limits.T_HeatSinkTemperature_Max := 150.0;
   Fluid.Limits.T_OilTemperature_Critical := 140.0;
   Fluid.Limits.T_OilSuperheat := 15.0;
   Fluid.Limits.T_CoolingSetpoint := 0.0;
   Fluid.T_AdditionalSuperHeatEvaporator := 8.0;
   Fluid.P_CriticalPoint := 3623.637;
   Compressor.CompressorTypeNumber := 1;
   Compressor.Limits.p_CrankCase_Max := 1600.0;
   Compressor.Limits.p_Oil_Min := 30.0;
   Compressor.Limits.n_Compressor_Max := 1200.0;
   Compressor.Limits.T_Motor_Max := 90.0;
   Compressor.Limits.M_Motor_Limit := 61.4;
   Compressor.Limits.T_Inverter_Max := 60.0;
   Compressor.Constant.CompressionVolume_L := 16.4;
   Compressor.Constant.CompressionLostPerPressureRatio := 3.41;
   Compressor.Constant.PumpEfficinecy := 93.69;
   Compressor.Settings := FALSE;
   System.SystemTypeNumber := 2;
   System.Limits.T_SuperHeatCompressorIn_Min := 2.0;
   System.Limits.T_Housing_Max := 50.0;
   System.Limits.T_CoolingCycle_Max := 65.0;
   System.Limits.p_CompressorOut_Max := 2700.0;
   System.Limits.p_EvaporatorOut_Max := 1550.0;
   System.Constant := FALSE;
   System.Settings.CooliungPump_ReversedPWM := FALSE;
   System.Settings.MotorCooling_AirFanCooledCycle := FALSE;
   System.Settings.DoubleExpansionValves := TRUE;
   System.Settings.Reserve3 := FALSE;
   System.Settings.Reserve4 := FALSE;
   System.Settings.Reserve5 := FALSE;
   VariableSetting.SystemType := 2;   // 1 = Alpha-1, 2 = Alpha-2
   VariableSetting.CompressorType := 1;
   VariableSetting.FluidType := 2;
   VariableSetting.OilPreheating_acv := TRUE;
   VariableSetting.OilHeatSetpoint_min := 45.0;
   VariableSetting.EnableViaHMI := TRUE;
   VariableSetting.EnableViaApplication := TRUE;
   VariableSetting.SourceOkFromApplication := FALSE;
   VariableSetting.SinkOkFromApplication := FALSE;
   VariableSetting.HeatSourceExternalControl := TRUE;
   VariableSetting.HeatSinkExternalControl := TRUE;
   StaticSetting.AdditionalSuperHeatOnColdStart := 0.0;
   StaticSetting.Limits.T_Ambient_Max := 40.0;
   StaticSetting.Limits.T_Cabinet_Max := 45.0;
END_DATA_BLOCK

DATA_BLOCK "Initialise_DB"   // DB36
AUTHOR : Heaten
VERSION : 0.1
// stored: AutoNumber true, DBAccessibleFromOPCUA true, DBAccessibleFromWebserver true, InstanceOfName Initialise, InstanceOfType FB
"Initialise"
BEGIN
END_DATA_BLOCK

DATA_BLOCK "InputProcessing_DB"   // DB47
AUTHOR : Heaten
VERSION : 0.1
// stored: AutoNumber true, DBAccessibleFromOPCUA true, DBAccessibleFromWebserver true, InstanceOfName InputProcessing, InstanceOfType FB
"InputProcessing"
BEGIN
END_DATA_BLOCK

DATA_BLOCK "InputWarningHandling_DB"   // DB10
AUTHOR : Heaten
VERSION : 0.1
// stored: AutoNumber true, DBAccessibleFromOPCUA true, DBAccessibleFromWebserver true, InstanceOfName InputWarningHandling, InstanceOfType FB
"InputWarningHandling"
BEGIN
END_DATA_BLOCK

DATA_BLOCK "OutputProcessing_DB"   // DB17
VERSION : 0.1
// stored: AutoNumber true, DBAccessibleFromOPCUA true, DBAccessibleFromWebserver true, InstanceOfName OutputProcessing, InstanceOfType FB
"OutputProcessing"
BEGIN
END_DATA_BLOCK

DATA_BLOCK "AlarmManagement_DB"   // DB23
VERSION : 0.1
// stored: AutoNumber true, DBAccessibleFromOPCUA true, DBAccessibleFromWebserver true, InstanceOfName AlarmManagement, InstanceOfType FB
"AlarmManagement"
BEGIN
END_DATA_BLOCK

DATA_BLOCK "Diagnosis_DB"   // DB1
VERSION : 0.1
// stored: AutoNumber true, DBAccessibleFromOPCUA true, DBAccessibleFromWebserver true, InstanceOfName Diagnosis, InstanceOfType FB
"Diagnosis"
BEGIN
END_DATA_BLOCK

DATA_BLOCK "HMI-Communication_DB"   // DB3
VERSION : 0.1
// stored: AutoNumber true, DBAccessibleFromOPCUA true, DBAccessibleFromWebserver true, InstanceOfName HMI-Communication, InstanceOfType FB
"HMI-Communication"
BEGIN
END_DATA_BLOCK

DATA_BLOCK "ApplicationCommunication_DB"   // DB11
VERSION : 0.1
// stored: AutoNumber true, DBAccessibleFromOPCUA true, DBAccessibleFromWebserver true, InstanceOfName ApplicationCommunication, InstanceOfType FB
"ApplicationCommunication"
BEGIN
END_DATA_BLOCK

